LIN {X 0,Y 354.792,Z 356.911,A -85,B 0,C 180,E1 -13288.404,E2 -13288.404} C_VEL
LIN {X 0,Y 354.852,Z 356.899,A -85,B 0,C 180,E1 -13291.619,E2 -13291.619} C_VEL
LIN {X 0,Y 354.898,Z 356.892,A -85,B 0,C 180,E1 -13294.172,E2 -13294.172} C_VEL
LIN {X 0,Y 354.833,Z 356.903,A -85,B 0,C 180,E1 -13297.894,E2 -13297.894} C_VEL
LIN {X 0,Y 354.92,Z 356.896,A -85,B 0,C 180,E1 -13301.891,E2 -13301.891} C_VEL
LIN {X 0,Y 354.941,Z 356.88,A -85,B 0,C 180,E1 -13305.98,E2 -13305.98} C_VEL
LIN {X 0,Y 354.981,Z 356.892,A -85,B 0,C 180,E1 -13309.736,E2 -13309.736} C_VEL
LIN {X 0,Y 355.112,Z 356.874,A -85,B 0,C 180,E1 -13312.037,E2 -13312.037} C_VEL
LIN {X 0,Y 355.091,Z 356.88,A -85,B 0,C 180,E1 -13314.321,E2 -13314.321} C_VEL
LIN {X 0,Y 355.244,Z 356.86,A -85,B 0,C 180,E1 -13317.732,E2 -13317.732} C_VEL
LIN {X 0,Y 355.395,Z 356.843,A -85,B 0,C 180,E1 -13320,E2 -13320} C_VEL
LIN {X 0,Y 355.244,Z 356.859,A -85,B 0,C 180,E1 -13322.267,E2 -13322.267} C_VEL
LIN {X 0,Y 355.136,Z 356.874,A -85,B 0,C 180,E1 -13326.819,E2 -13326.819} C_VEL
LIN {X 0,Y 355.013,Z 356.89,A -85,B 0,C 180,E1 -13329.112,E2 -13329.112} C_VEL
LIN {X 0,Y 354.919,Z 356.896,A -85,B 0,C 180,E1 -13332.581,E2 -13332.581} C_VEL
LIN {X 0,Y 354.887,Z 356.902,A -85,B 0,C 180,E1 -13336.096,E2 -13336.096} C_VEL
LIN {X 0,Y 354.904,Z 356.9,A -85,B 0,C 180,E1 -13338.472,E2 -13338.472} C_VEL
LIN {X 0,Y 354.832,Z 356.911,A -85,B 0,C 180,E1 -13342.106,E2 -13342.106} C_VEL
LIN {X 0,Y 354.897,Z 356.906,A -85,B 0,C 180,E1 -13345.827,E2 -13345.827} C_VEL
LIN {X 0,Y 354.852,Z 356.911,A -85,B 0,C 180,E1 -13349.679,E2 -13349.679} C_VEL
LIN {X 0,Y 354.803,Z 356.914,A -85,B 0,C 180,E1 -13353.702,E2 -13353.702} C_VEL
LIN {X 0,Y 354.851,Z 357.111,A -85,B 0,C 180,E1 -13355.707,E2 -13355.707} C_VEL
LIN {X 0,Y 355.545,Z 361.082,A -85,B 0,C 180,E1 -13359.238,E2 -13359.238} C_VEL
LIN {X 0,Y 356.332,Z 365.897,A -85,B 0,C 180,E1 -13363.135,E2 -13363.135} C_VEL
LIN {X 0,Y 357.017,Z 370.347,A -85,B 0,C 180,E1 -13366.451,E2 -13366.451} C_VEL
LIN {X 0,Y 357.144,Z 373.14,A -85,B 0,C 180,E1 -13368.398,E2 -13368.398} C_VEL
LIN {X 0,Y 356.7,Z 376.988,A -85,B 0,C 180,E1 -13370.914,E2 -13370.914} C_VEL
LIN {X 0,Y 356.204,Z 381.837,A -85,B 0,C 180,E1 -13373.992,E2 -13373.992} C_VEL
LIN {X 0,Y 355.641,Z 386.853,A -85,B 0,C 180,E1 -13377.082,E2 -13377.082} C_VEL
LIN {X 0,Y 354.999,Z 392.89,A -85,B 0,C 180,E1 -13380.747,E2 -13380.747} C_VEL
LIN {X 0,Y 356.577,Z 398.562,A -85,B 0,C 180,E1 -13381.035,E2 -13381.035} C_VEL
LIN {X 0,Y 360.847,Z 413.008,A -85,B 0,C 180,E1 -13381.89,E2 -13381.89} C_VEL
LIN {X 0,Y 364.022,Z 427.002,A -85,B 0,C 180,E1 -13382.822,E2 -13382.822} C_VEL
LIN {X 0,Y 366.355,Z 441.422,A -85,B 0,C 180,E1 -13383.916,E2 -13383.916} C_VEL
LIN {X 0,Y 366.773,Z 446.491,A -85,B 0,C 180,E1 -13384.331,E2 -13384.331} C_VEL
LIN {X 0,Y 365.079,Z 460.119,A -85,B 0,C 180,E1 -13385.4,E2 -13385.4} C_VEL
LIN {X 0,Y 363.21,Z 472.884,A -85,B 0,C 180,E1 -13386.63,E2 -13386.63} C_VEL
LIN {X 0,Y 361.147,Z 485.804,A -85,B 0,C 180,E1 -13388.151,E2 -13388.151} C_VEL
LIN {X 0,Y 359.279,Z 497.794,A -85,B 0,C 180,E1 -13389.875,E2 -13389.875} C_VEL
LIN {X 0,Y 357.694,Z 508.176,A -85,B 0,C 180,E1 -13391.678,E2 -13391.678} C_VEL
LIN {X 0,Y 356.178,Z 517.746,A -85,B 0,C 180,E1 -13393.67,E2 -13393.67} C_VEL
LIN {X 0,Y 355.076,Z 525.736,A -85,B 0,C 180,E1 -13395.677,E2 -13395.677} C_VEL
LIN {X 0,Y 354.215,Z 533.203,A -85,B 0,C 180,E1 -13397.976,E2 -13397.976} C_VEL
LIN {X 0,Y 353.613,Z 539.134,A -85,B 0,C 180,E1 -13400.275,E2 -13400.275} C_VEL
LIN {X 0,Y 353.433,Z 542.669,A -85,B 0,C 180,E1 -13401.999,E2 -13401.999} C_VEL
LIN {X 0,Y 353.28,Z 546.243,A -85,B 0,C 180,E1 -13404.292,E2 -13404.292} C_VEL
LIN {X 0,Y 353.246,Z 548.596,A -85,B 0,C 180,E1 -13406.579,E2 -13406.579} C_VEL
LIN {X 0,Y 353.373,Z 549.786,A -85,B 0,C 180,E1 -13408.861,E2 -13408.861} C_VEL
LIN {X 0,Y 353.373,Z 549.784,A -85,B 0,C 180,E1 -13411.14,E2 -13411.14} C_VEL
LIN {X 0,Y 353.25,Z 548.585,A -85,B 0,C 180,E1 -13413.422,E2 -13413.422} C_VEL
LIN {X 0,Y 353.33,Z 546.227,A -85,B 0,C 180,E1 -13415.708,E2 -13415.708} C_VEL
LIN {X 0,Y 353.435,Z 542.651,A -85,B 0,C 180,E1 -13418.002,E2 -13418.002} C_VEL
LIN {X 0,Y 353.692,Z 537.771,A -85,B 0,C 180,E1 -13420.302,E2 -13420.302} C_VEL
LIN {X 0,Y 354.381,Z 531.47,A -85,B 0,C 180,E1 -13422.601,E2 -13422.601} C_VEL
LIN {X 0,Y 355.367,Z 523.568,A -85,B 0,C 180,E1 -13424.898,E2 -13424.898} C_VEL
LIN {X 0,Y 356.555,Z 515.174,A -85,B 0,C 180,E1 -13426.902,E2 -13426.902} C_VEL
LIN {X 0,Y 358.192,Z 505.081,A -85,B 0,C 180,E1 -13428.89,E2 -13428.89} C_VEL
LIN {X 0,Y 359.777,Z 494.765,A -85,B 0,C 180,E1 -13430.587,E2 -13430.587} C_VEL
LIN {X 0,Y 361.699,Z 482.486,A -85,B 0,C 180,E1 -13432.266,E2 -13432.266} C_VEL
LIN {X 0,Y 363.774,Z 468.83,A -85,B 0,C 180,E1 -13433.785,E2 -13433.785} C_VEL
LIN {X 0,Y 365.735,Z 455.151,A -85,B 0,C 180,E1 -13435.009,E2 -13435.009} C_VEL
LIN {X 0,Y 366.764,Z 445.121,A -85,B 0,C 180,E1 -13435.76,E2 -13435.76} C_VEL
LIN {X 0,Y 364.758,Z 431.05,A -85,B 0,C 180,E1 -13436.869,E2 -13436.869} C_VEL
LIN {X 0,Y 361.626,Z 416.135,A -85,B 0,C 180,E1 -13437.898,E2 -13437.898} C_VEL
LIN {X 0,Y 357.697,Z 401.937,A -85,B 0,C 180,E1 -13438.761,E2 -13438.761} C_VEL
LIN {X 0,Y 355.006,Z 392.859,A -85,B 0,C 180,E1 -13439.255,E2 -13439.255} C_VEL
LIN {X 0,Y 355.62,Z 386.82,A -85,B 0,C 180,E1 -13442.921,E2 -13442.921} C_VEL
LIN {X 0,Y 356.167,Z 381.789,A -85,B 0,C 180,E1 -13445.999,E2 -13445.999} C_VEL
LIN {X 0,Y 356.829,Z 375.826,A -85,B 0,C 180,E1 -13449.814,E2 -13449.814} C_VEL
LIN {X 0,Y 357.151,Z 372.485,A -85,B 0,C 180,E1 -13451.994,E2 -13451.994} C_VEL
LIN {X 0,Y 356.778,Z 368.497,A -85,B 0,C 180,E1 -13454.835,E2 -13454.835} C_VEL
LIN {X 0,Y 356.1,Z 364.541,A -85,B 0,C 180,E1 -13457.854,E2 -13457.854} C_VEL
LIN {X 0,Y 355.553,Z 361.02,A -85,B 0,C 180,E1 -13460.764,E2 -13460.764} C_VEL
LIN {X 0,Y 354.841,Z 356.914,A -85,B 0,C 180,E1 -13464.509,E2 -13464.509} C_VEL
LIN {X 0,Y 354.789,Z 356.916,A -85,B 0,C 180,E1 -13467.667,E2 -13467.667} C_VEL
LIN {X 0,Y 354.849,Z 356.91,A -85,B 0,C 180,E1 -13471.619,E2 -13471.619} C_VEL
LIN {X 0,Y 354.902,Z 356.905,A -85,B 0,C 180,E1 -13474.173,E2 -13474.173} C_VEL
LIN {X 0,Y 354.837,Z 356.911,A -85,B 0,C 180,E1 -13477.894,E2 -13477.894} C_VEL
LIN {X 0,Y 354.926,Z 356.901,A -85,B 0,C 180,E1 -13481.892,E2 -13481.892} C_VEL
LIN {X 0,Y 354.946,Z 356.901,A -85,B 0,C 180,E1 -13485.981,E2 -13485.981} C_VEL
LIN {X 0,Y 354.981,Z 356.895,A -85,B 0,C 180,E1 -13489.736,E2 -13489.736} C_VEL
LIN {X 0,Y 355.118,Z 356.879,A -85,B 0,C 180,E1 -13492.037,E2 -13492.037} C_VEL
LIN {X 0,Y 355.096,Z 356.878,A -85,B 0,C 180,E1 -13494.321,E2 -13494.321} C_VEL
LIN {X 0,Y 355.249,Z 356.858,A -85,B 0,C 180,E1 -13497.733,E2 -13497.733} C_VEL
LIN {X 0,Y 355.399,Z 356.838,A -85,B 0,C 180,E1 -13500,E2 -13500} C_VEL
LIN {X 0,Y 355.249,Z 356.858,A -85,B 0,C 180,E1 -13502.268,E2 -13502.268} C_VEL
LIN {X 0,Y 355.142,Z 356.868,A -85,B 0,C 180,E1 -13506.819,E2 -13506.819} C_VEL
LIN {X 0,Y 355.019,Z 356.888,A -85,B 0,C 180,E1 -13509.112,E2 -13509.112} C_VEL
LIN {X 0,Y 354.924,Z 356.873,A -85,B 0,C 180,E1 -13512.581,E2 -13512.581} C_VEL
LIN {X 0,Y 354.893,Z 356.901,A -85,B 0,C 180,E1 -13516.096,E2 -13516.096} C_VEL
LIN {X 0,Y 354.905,Z 356.894,A -85,B 0,C 180,E1 -13518.472,E2 -13518.472} C_VEL
LIN {X 0,Y 354.83,Z 356.902,A -85,B 0,C 180,E1 -13522.106,E2 -13522.106} C_VEL
LIN {X 0,Y 354.902,Z 356.893,A -85,B 0,C 180,E1 -13525.827,E2 -13525.827} C_VEL
LIN {X 0,Y 354.821,Z 356.91,A -85,B 0,C 180,E1 -13529.682,E2 -13529.682} C_VEL
LIN {X 0,Y 354.809,Z 356.9,A -85,B 0,C 180,E1 -13533.702,E2 -13533.702} C_VEL
LIN {X 0,Y 354.802,Z 356.917,A -85,B 0,C 180,E1 -13536.459,E2 -13536.459} C_VEL
LIN {X 0,Y 354.827,Z 356.912,A -85,B 0,C 180,E1 -13539.423,E2 -13539.423} C_VEL
LIN {X 0,Y 354.791,Z 356.918,A -85,B 0,C 180,E1 -13542.867,E2 -13542.867} C_VEL
LIN {X 0,Y 354.759,Z 356.925,A -85,B 0,C 180,E1 -13546.102,E2 -13546.102} C_VEL
LIN {X 0,Y 354.646,Z 356.938,A -85,B 0,C 180,E1 -13549.159,E2 -13549.159} C_VEL
LIN {X 0,Y 354.551,Z 356.949,A -85,B 0,C 180,E1 -13550.63,E2 -13550.63} C_VEL
LIN {X 0,Y 354.388,Z 358.655,A -85,B 0,C 180,E1 -13553.491,E2 -13553.491} C_VEL
LIN {X 0,Y 354.329,Z 360.804,A -85,B 0,C 180,E1 -13556.414,E2 -13556.414} C_VEL
LIN {X 0,Y 354.246,Z 362.804,A -85,B 0,C 180,E1 -13558.947,E2 -13558.947} C_VEL
LIN {X 0,Y 354.18,Z 364.301,A -85,B 0,C 180,E1 -13560.767,E2 -13560.767} C_VEL
LIN {X 0,Y 355.13,Z 367.269,A -85,B 0,C 180,E1 -13560.946,E2 -13560.946} C_VEL
LIN {X 0,Y 360.606,Z 380.429,A -85,B 0,C 180,E1 -13561.869,E2 -13561.869} C_VEL
LIN {X 0,Y 365.001,Z 393.413,A -85,B 0,C 180,E1 -13562.86,E2 -13562.86} C_VEL
LIN {X 0,Y 368.598,Z 406.777,A -85,B 0,C 180,E1 -13563.989,E2 -13563.989} C_VEL
LIN {X 0,Y 367.247,Z 420.846,A -85,B 0,C 180,E1 -13564.996,E2 -13564.996} C_VEL
LIN {X 0,Y 365.75,Z 432.854,A -85,B 0,C 180,E1 -13566.051,E2 -13566.051} C_VEL
LIN {X 0,Y 363.869,Z 445.767,A -85,B 0,C 180,E1 -13567.425,E2 -13567.425} C_VEL
LIN {X 0,Y 362.072,Z 457.604,A -85,B 0,C 180,E1 -13568.965,E2 -13568.965} C_VEL
LIN {X 0,Y 360.34,Z 468.309,A -85,B 0,C 180,E1 -13570.636,E2 -13570.636} C_VEL
LIN {X 0,Y 358.782,Z 477.435,A -85,B 0,C 180,E1 -13572.324,E2 -13572.324} C_VEL
LIN {X 0,Y 357.29,Z 486.251,A -85,B 0,C 180,E1 -13574.283,E2 -13574.283} C_VEL
LIN {X 0,Y 356.202,Z 493.723,A -85,B 0,C 180,E1 -13576.304,E2 -13576.304} C_VEL
LIN {X 0,Y 355.03,Z 500.622,A -85,B 0,C 180,E1 -13578.582,E2 -13578.582} C_VEL
LIN {X 0,Y 354.333,Z 506.03,A -85,B 0,C 180,E1 -13580.869,E2 -13580.869} C_VEL
LIN {X 0,Y 353.792,Z 510.388,A -85,B 0,C 180,E1 -13583.335,E2 -13583.335} C_VEL
LIN {X 0,Y 353.521,Z 512.977,A -85,B 0,C 180,E1 -13585.439,E2 -13585.439} C_VEL
LIN {X 0,Y 353.488,Z 514.694,A -85,B 0,C 180,E1 -13587.721,E2 -13587.721} C_VEL
LIN {X 0,Y 353.421,Z 515.297,A -85,B 0,C 180,E1 -13590,E2 -13590} C_VEL
LIN {X 0,Y 353.488,Z 514.739,A -85,B 0,C 180,E1 -13592.278,E2 -13592.278} C_VEL
LIN {X 0,Y 353.52,Z 513.08,A -85,B 0,C 180,E1 -13594.561,E2 -13594.561} C_VEL
LIN {X 0,Y 353.803,Z 510.271,A -85,B 0,C 180,E1 -13596.845,E2 -13596.845} C_VEL
LIN {X 0,Y 354.289,Z 506.244,A -85,B 0,C 180,E1 -13599.131,E2 -13599.131} C_VEL
LIN {X 0,Y 354.996,Z 500.903,A -85,B 0,C 180,E1 -13601.418,E2 -13601.418} C_VEL
LIN {X 0,Y 356.098,Z 494.084,A -85,B 0,C 180,E1 -13603.699,E2 -13603.699} C_VEL
LIN {X 0,Y 357.197,Z 486.711,A -85,B 0,C 180,E1 -13605.707,E2 -13605.707} C_VEL
LIN {X 0,Y 358.711,Z 477.904,A -85,B 0,C 180,E1 -13607.678,E2 -13607.678} C_VEL
LIN {X 0,Y 360.259,Z 468.873,A -85,B 0,C 180,E1 -13609.368,E2 -13609.368} C_VEL
LIN {X 0,Y 362.038,Z 457.697,A -85,B 0,C 180,E1 -13611.126,E2 -13611.126} C_VEL
LIN {X 0,Y 363.94,Z 445.402,A -85,B 0,C 180,E1 -13612.719,E2 -13612.719} C_VEL
LIN {X 0,Y 365.804,Z 432.419,A -85,B 0,C 180,E1 -13614.095,E2 -13614.095} C_VEL
LIN {X 0,Y 367.449,Z 419.304,A -85,B 0,C 180,E1 -13615.226,E2 -13615.226} C_VEL
LIN {X 0,Y 368.586,Z 406.514,A -85,B 0,C 180,E1 -13616.133,E2 -13616.133} C_VEL
LIN {X 0,Y 364.62,Z 392.07,A -85,B 0,C 180,E1 -13617.345,E2 -13617.345} C_VEL
LIN {X 0,Y 359.758,Z 378.332,A -85,B 0,C 180,E1 -13618.393,E2 -13618.393} C_VEL
LIN {X 0,Y 354.941,Z 366.959,A -85,B 0,C 180,E1 -13619.187,E2 -13619.187} C_VEL
LIN {X 0,Y 354.127,Z 364.27,A -85,B 0,C 180,E1 -13619.354,E2 -13619.354} C_VEL
LIN {X 0,Y 354.277,Z 361.813,A -85,B 0,C 180,E1 -13622.385,E2 -13622.385} C_VEL
LIN {X 0,Y 354.282,Z 361.372,A -85,B 0,C 180,E1 -13622.97,E2 -13622.97} C_VEL
LIN {X 0,Y 353.664,Z 360.751,A -85,B 0,C 180,E1 -13623.914,E2 -13623.914} C_VEL
LIN {X 0,Y 350.891,Z 359.984,A -85,B 0,C 180,E1 -13625.456,E2 -13625.456} C_VEL
LIN {X 0,Y 348.521,Z 359.395,A -85,B 0,C 180,E1 -13626.703,E2 -13626.703} C_VEL
LIN {X 0,Y 347.502,Z 358.841,A -85,B 0,C 180,E1 -13627.666,E2 -13627.666} C_VEL
LIN {X 0,Y 347.418,Z 358.622,A -85,B 0,C 180,E1 -13627.991,E2 -13627.991} C_VEL
LIN {X 0,Y 347.444,Z 358.029,A -85,B 0,C 180,E1 -13628.833,E2 -13628.833} C_VEL
LIN {X 0,Y 347.67,Z 357.799,A -85,B 0,C 180,E1 -13631.841,E2 -13631.841} C_VEL
LIN {X 0,Y 347.702,Z 357.799,A -85,B 0,C 180,E1 -13635.027,E2 -13635.027} C_VEL
LIN {X 0,Y 347.749,Z 357.793,A -85,B 0,C 180,E1 -13638.397,E2 -13638.397} C_VEL
LIN {X 0,Y 347.773,Z 357.791,A -85,B 0,C 180,E1 -13642.011,E2 -13642.011} C_VEL
LIN {X 0,Y 347.743,Z 357.789,A -85,B 0,C 180,E1 -13645.536,E2 -13645.536} C_VEL
LIN {X 0,Y 347.762,Z 357.793,A -85,B 0,C 180,E1 -13649.653,E2 -13649.653} C_VEL
LIN {X 0,Y 347.851,Z 357.763,A -85,B 0,C 180,E1 -13652.744,E2 -13652.744} C_VEL
LIN {X 0,Y 347.787,Z 357.788,A -85,B 0,C 180,E1 -13656.162,E2 -13656.162} C_VEL
LIN {X 0,Y 347.81,Z 357.764,A -85,B 0,C 180,E1 -13659.909,E2 -13659.909} C_VEL
LIN {X 0,Y 347.864,Z 357.778,A -85,B 0,C 180,E1 -13662.359,E2 -13662.359} C_VEL
LIN {X 0,Y 347.895,Z 357.757,A -85,B 0,C 180,E1 -13665.971,E2 -13665.971} C_VEL
LIN {X 0,Y 347.931,Z 357.767,A -85,B 0,C 180,E1 -13669.526,E2 -13669.526} C_VEL
LIN {X 0,Y 348.072,Z 357.751,A -85,B 0,C 180,E1 -13671.875,E2 -13671.875} C_VEL
LIN {X 0,Y 348.066,Z 357.755,A -85,B 0,C 180,E1 -13674.206,E2 -13674.206} C_VEL
LIN {X 0,Y 348.206,Z 357.737,A -85,B 0,C 180,E1 -13677.686,E2 -13677.686} C_VEL
LIN {X 0,Y 348.365,Z 357.719,A -85,B 0,C 180,E1 -13680,E2 -13680} C_VEL
LIN {X 0,Y 348.207,Z 357.736,A -85,B 0,C 180,E1 -13682.313,E2 -13682.313} C_VEL
LIN {X 0,Y 348.104,Z 357.749,A -85,B 0,C 180,E1 -13686.958,E2 -13686.958} C_VEL
LIN {X 0,Y 347.965,Z 357.769,A -85,B 0,C 180,E1 -13689.298,E2 -13689.298} C_VEL
LIN {X 0,Y 347.888,Z 357.772,A -85,B 0,C 180,E1 -13692.839,E2 -13692.839} C_VEL
LIN {X 0,Y 347.837,Z 357.78,A -85,B 0,C 180,E1 -13696.431,E2 -13696.431} C_VEL
LIN {X 0,Y 347.853,Z 357.78,A -85,B 0,C 180,E1 -13698.86,E2 -13698.86} C_VEL
LIN {X 0,Y 347.772,Z 357.791,A -85,B 0,C 180,E1 -13702.579,E2 -13702.579} C_VEL
LIN {X 0,Y 347.81,Z 357.788,A -85,B 0,C 180,E1 -13705.108,E2 -13705.108} C_VEL
LIN {X 0,Y 347.81,Z 357.79,A -85,B 0,C 180,E1 -13707.694,E2 -13707.694} C_VEL
LIN {X 0,Y 347.762,Z 357.794,A -85,B 0,C 180,E1 -13710.347,E2 -13710.347} C_VEL
LIN {X 0,Y 347.742,Z 357.797,A -85,B 0,C 180,E1 -13714.464,E2 -13714.464} C_VEL
LIN {X 0,Y 347.821,Z 357.98,A -85,B 0,C 180,E1 -13715.16,E2 -13715.16} C_VEL
LIN {X 0,Y 348.464,Z 361.88,A -85,B 0,C 180,E1 -13718.698,E2 -13718.698} C_VEL
LIN {X 0,Y 349.074,Z 365.588,A -85,B 0,C 180,E1 -13721.848,E2 -13721.848} C_VEL
LIN {X 0,Y 349.84,Z 370.026,A -85,B 0,C 180,E1 -13725.323,E2 -13725.323} C_VEL
LIN {X 0,Y 350.146,Z 373.663,A -85,B 0,C 180,E1 -13727.958,E2 -13727.958} C_VEL
LIN {X 0,Y 349.709,Z 377.764,A -85,B 0,C 180,E1 -13730.726,E2 -13730.726} C_VEL
LIN {X 0,Y 349.092,Z 383.238,A -85,B 0,C 180,E1 -13734.28,E2 -13734.28} C_VEL
LIN {X 0,Y 348.473,Z 388.953,A -85,B 0,C 180,E1 -13737.893,E2 -13737.893} C_VEL
LIN {X 0,Y 348.058,Z 392.505,A -85,B 0,C 180,E1 -13740.097,E2 -13740.097} C_VEL
LIN {X 0,Y 348.978,Z 395.921,A -85,B 0,C 180,E1 -13740.281,E2 -13740.281} C_VEL
LIN {X 0,Y 353.632,Z 411.282,A -85,B 0,C 180,E1 -13741.205,E2 -13741.205} C_VEL
LIN {X 0,Y 357.038,Z 425.815,A -85,B 0,C 180,E1 -13742.197,E2 -13742.197} C_VEL
LIN {X 0,Y 359.373,Z 439.628,A -85,B 0,C 180,E1 -13743.27,E2 -13743.27} C_VEL
LIN {X 0,Y 360.234,Z 446.964,A -85,B 0,C 180,E1 -13743.894,E2 -13743.894} C_VEL
LIN {X 0,Y 358.379,Z 461.362,A -85,B 0,C 180,E1 -13745.063,E2 -13745.063} C_VEL
LIN {X 0,Y 356.448,Z 473.835,A -85,B 0,C 180,E1 -13746.314,E2 -13746.314} C_VEL
LIN {X 0,Y 354.316,Z 486.533,A -85,B 0,C 180,E1 -13747.86,E2 -13747.86} C_VEL
LIN {X 0,Y 352.389,Z 498.32,A -85,B 0,C 180,E1 -13749.613,E2 -13749.613} C_VEL
LIN {X 0,Y 350.889,Z 507.826,A -85,B 0,C 180,E1 -13751.309,E2 -13751.309} C_VEL
LIN {X 0,Y 349.288,Z 517.396,A -85,B 0,C 180,E1 -13753.339,E2 -13753.339} C_VEL
LIN {X 0,Y 348.092,Z 525.588,A -85,B 0,C 180,E1 -13755.442,E2 -13755.442} C_VEL
LIN {X 0,Y 347.202,Z 532.853,A -85,B 0,C 180,E1 -13757.729,E2 -13757.729} C_VEL
LIN {X 0,Y 346.555,Z 538.784,A -85,B 0,C 180,E1 -13760.074,E2 -13760.074} C_VEL
LIN {X 0,Y 346.358,Z 542.32,A -85,B 0,C 180,E1 -13761.835,E2 -13761.835} C_VEL
LIN {X 0,Y 346.199,Z 545.895,A -85,B 0,C 180,E1 -13764.175,E2 -13764.175} C_VEL
LIN {X 0,Y 346.168,Z 548.249,A -85,B 0,C 180,E1 -13766.509,E2 -13766.509} C_VEL
LIN {X 0,Y 346.276,Z 549.438,A -85,B 0,C 180,E1 -13768.838,E2 -13768.838} C_VEL
LIN {X 0,Y 346.276,Z 549.436,A -85,B 0,C 180,E1 -13771.163,E2 -13771.163} C_VEL
LIN {X 0,Y 346.172,Z 548.237,A -85,B 0,C 180,E1 -13773.492,E2 -13773.492} C_VEL
LIN {X 0,Y 346.286,Z 545.621,A -85,B 0,C 180,E1 -13776.028,E2 -13776.028} C_VEL
LIN {X 0,Y 346.418,Z 541.213,A -85,B 0,C 180,E1 -13778.752,E2 -13778.752} C_VEL
LIN {X 0,Y 346.835,Z 535.971,A -85,B 0,C 180,E1 -13781.099,E2 -13781.099} C_VEL
LIN {X 0,Y 347.596,Z 529.278,A -85,B 0,C 180,E1 -13783.446,E2 -13783.446} C_VEL
LIN {X 0,Y 348.579,Z 522.082,A -85,B 0,C 180,E1 -13785.495,E2 -13785.495} C_VEL
LIN {X 0,Y 349.86,Z 513.45,A -85,B 0,C 180,E1 -13787.537,E2 -13787.537} C_VEL
LIN {X 0,Y 351.651,Z 503.082,A -85,B 0,C 180,E1 -13789.558,E2 -13789.558} C_VEL
LIN {X 0,Y 353.364,Z 492.483,A -85,B 0,C 180,E1 -13791.283,E2 -13791.283} C_VEL
LIN {X 0,Y 355.241,Z 480.973,A -85,B 0,C 180,E1 -13792.846,E2 -13792.846} C_VEL
LIN {X 0,Y 357.257,Z 468.476,A -85,B 0,C 180,E1 -13794.246,E2 -13794.246} C_VEL
LIN {X 0,Y 359.281,Z 454.797,A -85,B 0,C 180,E1 -13795.49,E2 -13795.49} C_VEL
LIN {X 0,Y 360.162,Z 446.23,A -85,B 0,C 180,E1 -13796.153,E2 -13796.153} C_VEL
LIN {X 0,Y 358.311,Z 432.718,A -85,B 0,C 180,E1 -13797.27,E2 -13797.27} C_VEL
LIN {X 0,Y 355.067,Z 416.892,A -85,B 0,C 180,E1 -13798.41,E2 -13798.41} C_VEL
LIN {X 0,Y 350.843,Z 401.801,A -85,B 0,C 180,E1 -13799.37,E2 -13799.37} C_VEL
LIN {X 0,Y 348.151,Z 393.412,A -85,B 0,C 180,E1 -13799.842,E2 -13799.842} C_VEL
LIN {X 0,Y 348.047,Z 392.512,A -85,B 0,C 180,E1 -13799.884,E2 -13799.884} C_VEL
LIN {X 0,Y 348.861,Z 385.406,A -85,B 0,C 180,E1 -13804.314,E2 -13804.314} C_VEL
LIN {X 0,Y 349.519,Z 379.113,A -85,B 0,C 180,E1 -13808.354,E2 -13808.354} C_VEL
LIN {X 0,Y 350.121,Z 374.414,A -85,B 0,C 180,E1 -13811.485,E2 -13811.485} C_VEL
LIN {X 0,Y 350,Z 371.261,A -85,B 0,C 180,E1 -13813.707,E2 -13813.707} C_VEL
LIN {X 0,Y 349.36,Z 367.126,A -85,B 0,C 180,E1 -13816.845,E2 -13816.845} C_VEL
LIN {X 0,Y 348.741,Z 363.333,A -85,B 0,C 180,E1 -13819.978,E2 -13819.978} C_VEL
LIN {X 0,Y 347.99,Z 358.928,A -85,B 0,C 180,E1 -13823.886,E2 -13823.886} C_VEL
LIN {X 0,Y 347.78,Z 357.796,A -85,B 0,C 180,E1 -13825.189,E2 -13825.189} C_VEL
LIN {X 0,Y 347.747,Z 357.796,A -85,B 0,C 180,E1 -13828.301,E2 -13828.301} C_VEL
LIN {X 0,Y 347.781,Z 357.791,A -85,B 0,C 180,E1 -13830.988,E2 -13830.988} C_VEL
LIN {X 0,Y 347.834,Z 357.785,A -85,B 0,C 180,E1 -13833.608,E2 -13833.608} C_VEL
LIN {X 0,Y 347.791,Z 357.788,A -85,B 0,C 180,E1 -13836.162,E2 -13836.162} C_VEL
LIN {X 0,Y 347.82,Z 357.786,A -85,B 0,C 180,E1 -13839.91,E2 -13839.91} C_VEL
LIN {X 0,Y 347.869,Z 357.779,A -85,B 0,C 180,E1 -13842.36,E2 -13842.36} C_VEL
LIN {X 0,Y 347.9,Z 357.779,A -85,B 0,C 180,E1 -13845.971,E2 -13845.971} C_VEL
LIN {X 0,Y 347.932,Z 357.774,A -85,B 0,C 180,E1 -13849.526,E2 -13849.526} C_VEL
LIN {X 0,Y 348.078,Z 357.755,A -85,B 0,C 180,E1 -13851.875,E2 -13851.875} C_VEL
LIN {X 0,Y 348.071,Z 357.754,A -85,B 0,C 180,E1 -13854.206,E2 -13854.206} C_VEL
LIN {X 0,Y 348.211,Z 357.735,A -85,B 0,C 180,E1 -13857.687,E2 -13857.687} C_VEL
LIN {X 0,Y 348.348,Z 357.716,A -85,B 0,C 180,E1 -13860,E2 -13860} C_VEL
LIN {X 0,Y 348.211,Z 357.735,A -85,B 0,C 180,E1 -13862.314,E2 -13862.314} C_VEL
LIN {X 0,Y 348.11,Z 357.744,A -85,B 0,C 180,E1 -13866.958,E2 -13866.958} C_VEL
LIN {X 0,Y 347.971,Z 357.765,A -85,B 0,C 180,E1 -13869.299,E2 -13869.299} C_VEL
LIN {X 0,Y 347.893,Z 357.747,A -85,B 0,C 180,E1 -13872.839,E2 -13872.839} C_VEL
LIN {X 0,Y 347.843,Z 357.781,A -85,B 0,C 180,E1 -13876.431,E2 -13876.431} C_VEL
LIN {X 0,Y 347.854,Z 357.771,A -85,B 0,C 180,E1 -13878.86,E2 -13878.86} C_VEL
LIN {X 0,Y 347.771,Z 357.784,A -85,B 0,C 180,E1 -13882.58,E2 -13882.58} C_VEL
LIN {X 0,Y 347.815,Z 357.782,A -85,B 0,C 180,E1 -13885.108,E2 -13885.108} C_VEL
LIN {X 0,Y 347.811,Z 357.768,A -85,B 0,C 180,E1 -13887.694,E2 -13887.694} C_VEL
LIN {X 0,Y 347.752,Z 357.795,A -85,B 0,C 180,E1 -13890.348,E2 -13890.348} C_VEL
LIN {X 0,Y 347.751,Z 357.781,A -85,B 0,C 180,E1 -13894.044,E2 -13894.044} C_VEL
LIN {X 0,Y 347.766,Z 357.791,A -85,B 0,C 180,E1 -13897.32,E2 -13897.32} C_VEL
LIN {X 0,Y 347.736,Z 357.796,A -85,B 0,C 180,E1 -13900.297,E2 -13900.297} C_VEL
LIN {X 0,Y 347.726,Z 357.798,A -85,B 0,C 180,E1 -13903.408,E2 -13903.408} C_VEL
LIN {X 0,Y 347.718,Z 357.803,A -85,B 0,C 180,E1 -13906.688,E2 -13906.688} C_VEL
LIN {X 0,Y 347.551,Z 357.821,A -85,B 0,C 180,E1 -13909.677,E2 -13909.677} C_VEL
LIN {X 0,Y 347.443,Z 357.947,A -85,B 0,C 180,E1 -13911.166,E2 -13911.166} C_VEL
LIN {X 0,Y 347.335,Z 360.038,A -85,B 0,C 180,E1 -13914.07,E2 -13914.07} C_VEL
LIN {X 0,Y 347.266,Z 362.085,A -85,B 0,C 180,E1 -13916.877,E2 -13916.877} C_VEL
LIN {X 0,Y 347.132,Z 364.664,A -85,B 0,C 180,E1 -13920.105,E2 -13920.105} C_VEL
LIN {X 0,Y 348.332,Z 368.023,A -85,B 0,C 180,E1 -13920.333,E2 -13920.333} C_VEL
LIN {X 0,Y 353.964,Z 381.605,A -85,B 0,C 180,E1 -13921.328,E2 -13921.328} C_VEL
LIN {X 0,Y 358.362,Z 394.279,A -85,B 0,C 180,E1 -13922.34,E2 -13922.34} C_VEL
LIN {X 0,Y 361.801,Z 407.157,A -85,B 0,C 180,E1 -13923.463,E2 -13923.463} C_VEL
LIN {X 0,Y 362.156,Z 409.029,A -85,B 0,C 180,E1 -13923.623,E2 -13923.623} C_VEL
LIN {X 0,Y 360.697,Z 422.417,A -85,B 0,C 180,E1 -13924.617,E2 -13924.617} C_VEL
LIN {X 0,Y 359.104,Z 434.623,A -85,B 0,C 180,E1 -13925.733,E2 -13925.733} C_VEL
LIN {X 0,Y 357.148,Z 447.283,A -85,B 0,C 180,E1 -13927.129,E2 -13927.129} C_VEL
LIN {X 0,Y 355.539,Z 457.305,A -85,B 0,C 180,E1 -13928.456,E2 -13928.456} C_VEL
LIN {X 0,Y 353.901,Z 467.036,A -85,B 0,C 180,E1 -13929.966,E2 -13929.966} C_VEL
LIN {X 0,Y 351.994,Z 477.787,A -85,B 0,C 180,E1 -13931.972,E2 -13931.972} C_VEL
LIN {X 0,Y 350.429,Z 486.674,A -85,B 0,C 180,E1 -13933.985,E2 -13933.985} C_VEL
LIN {X 0,Y 349.268,Z 494.075,A -85,B 0,C 180,E1 -13936.026,E2 -13936.026} C_VEL
LIN {X 0,Y 348.053,Z 500.972,A -85,B 0,C 180,E1 -13938.35,E2 -13938.35} C_VEL
LIN {X 0,Y 347.309,Z 506.38,A -85,B 0,C 180,E1 -13940.683,E2 -13940.683} C_VEL
LIN {X 0,Y 346.717,Z 510.939,A -85,B 0,C 180,E1 -13943.333,E2 -13943.333} C_VEL
LIN {X 0,Y 346.46,Z 513.325,A -85,B 0,C 180,E1 -13945.345,E2 -13945.345} C_VEL
LIN {X 0,Y 346.395,Z 515.042,A -85,B 0,C 180,E1 -13947.674,E2 -13947.674} C_VEL
LIN {X 0,Y 346.341,Z 515.644,A -85,B 0,C 180,E1 -13950,E2 -13950} C_VEL
LIN {X 0,Y 346.395,Z 515.086,A -85,B 0,C 180,E1 -13952.325,E2 -13952.325} C_VEL
LIN {X 0,Y 346.459,Z 513.427,A -85,B 0,C 180,E1 -13954.654,E2 -13954.654} C_VEL
LIN {X 0,Y 346.746,Z 510.618,A -85,B 0,C 180,E1 -13956.985,E2 -13956.985} C_VEL
LIN {X 0,Y 347.276,Z 506.591,A -85,B 0,C 180,E1 -13959.317,E2 -13959.317} C_VEL
LIN {X 0,Y 348.021,Z 501.25,A -85,B 0,C 180,E1 -13961.65,E2 -13961.65} C_VEL
LIN {X 0,Y 349.174,Z 494.431,A -85,B 0,C 180,E1 -13963.976,E2 -13963.976} C_VEL
LIN {X 0,Y 350.336,Z 487.102,A -85,B 0,C 180,E1 -13966.011,E2 -13966.011} C_VEL
LIN {X 0,Y 351.939,Z 478.25,A -85,B 0,C 180,E1 -13968.03,E2 -13968.03} C_VEL
LIN {X 0,Y 353.528,Z 469.22,A -85,B 0,C 180,E1 -13969.752,E2 -13969.752} C_VEL
LIN {X 0,Y 355.345,Z 458.483,A -85,B 0,C 180,E1 -13971.474,E2 -13971.474} C_VEL
LIN {X 0,Y 357.213,Z 446.911,A -85,B 0,C 180,E1 -13973.018,E2 -13973.018} C_VEL
LIN {X 0,Y 359.179,Z 434.176,A -85,B 0,C 180,E1 -13974.415,E2 -13974.415} C_VEL
LIN {X 0,Y 360.738,Z 422.41,A -85,B 0,C 180,E1 -13975.486,E2 -13975.486} C_VEL
LIN {X 0,Y 362.161,Z 408.662,A -85,B 0,C 180,E1 -13976.508,E2 -13976.508} C_VEL
LIN {X 0,Y 358.206,Z 393.724,A -85,B 0,C 180,E1 -13977.808,E2 -13977.808} C_VEL
LIN {X 0,Y 352.975,Z 379.129,A -85,B 0,C 180,E1 -13978.974,E2 -13978.974} C_VEL
LIN {X 0,Y 348.071,Z 367.614,A -85,B 0,C 180,E1 -13979.812,E2 -13979.812} C_VEL
LIN {X 0,Y 347.116,Z 364.65,A -85,B 0,C 180,E1 -13979.995,E2 -13979.995} C_VEL
LIN {X 0,Y 347.26,Z 362.175,A -85,B 0,C 180,E1 -13983.122,E2 -13983.122} C_VEL
LIN {X 0,Y 347.339,Z 360.094,A -85,B 0,C 180,E1 -13985.967,E2 -13985.967} C_VEL
LIN {X 0,Y 347.418,Z 358.622,A -85,B 0,C 180,E1 -13987.991,E2 -13987.991} C_VEL
LIN {X 0,Y 346.776,Z 358.196,A -85,B 0,C 180,E1 -13988.956,E2 -13988.956} C_VEL
LIN {X 0,Y 344.046,Z 358.252,A -85,B 0,C 180,E1 -13990.537,E2 -13990.537} C_VEL
LIN {X 0,Y 341.728,Z 358.539,A -85,B 0,C 180,E1 -13991.819,E2 -13991.819} C_VEL
LIN {X 0,Y 340.727,Z 358.665,A -85,B 0,C 180,E1 -13992.808,E2 -13992.808} C_VEL
LIN {X 0,Y 340.641,Z 358.675,A -85,B 0,C 180,E1 -13993.143,E2 -13993.143} C_VEL
LIN {X 0,Y 340.674,Z 358.675,A -85,B 0,C 180,E1 -13997.095,E2 -13997.095} C_VEL
LIN {X 0,Y 340.697,Z 358.672,A -85,B 0,C 180,E1 -14000.247,E2 -14000.247} C_VEL
LIN {X 0,Y 340.709,Z 358.67,A -85,B 0,C 180,E1 -14003.559,E2 -14003.559} C_VEL
LIN {X 0,Y 340.692,Z 358.662,A -85,B 0,C 180,E1 -14006.153,E2 -14006.153} C_VEL
LIN {X 0,Y 340.773,Z 358.661,A -85,B 0,C 180,E1 -14010.332,E2 -14010.332} C_VEL
LIN {X 0,Y 340.803,Z 358.641,A -85,B 0,C 180,E1 -14013.02,E2 -14013.02} C_VEL
LIN {X 0,Y 340.727,Z 358.667,A -85,B 0,C 180,E1 -14016.927,E2 -14016.927} C_VEL
LIN {X 0,Y 340.788,Z 358.645,A -85,B 0,C 180,E1 -14020.733,E2 -14020.733} C_VEL
LIN {X 0,Y 340.785,Z 358.661,A -85,B 0,C 180,E1 -14023.218,E2 -14023.218} C_VEL
LIN {X 0,Y 340.845,Z 358.629,A -85,B 0,C 180,E1 -14026.89,E2 -14026.89} C_VEL
LIN {X 0,Y 340.928,Z 358.643,A -85,B 0,C 180,E1 -14030.508,E2 -14030.508} C_VEL
LIN {X 0,Y 341.074,Z 358.626,A -85,B 0,C 180,E1 -14032.898,E2 -14032.898} C_VEL
LIN {X 0,Y 341.168,Z 358.614,A -85,B 0,C 180,E1 -14037.639,E2 -14037.639} C_VEL
LIN {X 0,Y 341.314,Z 358.597,A -85,B 0,C 180,E1 -14040,E2 -14040} C_VEL
LIN {X 0,Y 341.168,Z 358.612,A -85,B 0,C 180,E1 -14042.361,E2 -14042.361} C_VEL
LIN {X 0,Y 341.074,Z 358.625,A -85,B 0,C 180,E1 -14047.102,E2 -14047.102} C_VEL
LIN {X 0,Y 340.869,Z 358.651,A -85,B 0,C 180,E1 -14050.694,E2 -14050.694} C_VEL
LIN {X 0,Y 340.86,Z 358.65,A -85,B 0,C 180,E1 -14054.325,E2 -14054.325} C_VEL
LIN {X 0,Y 340.835,Z 358.652,A -85,B 0,C 180,E1 -14058.467,E2 -14058.467} C_VEL
LIN {X 0,Y 340.751,Z 358.666,A -85,B 0,C 180,E1 -14061.857,E2 -14061.857} C_VEL
LIN {X 0,Y 340.77,Z 358.665,A -85,B 0,C 180,E1 -14065.664,E2 -14065.664} C_VEL
LIN {X 0,Y 340.74,Z 358.669,A -85,B 0,C 180,E1 -14068.32,E2 -14068.32} C_VEL
LIN {X 0,Y 340.702,Z 358.673,A -85,B 0,C 180,E1 -14071.044,E2 -14071.044} C_VEL
LIN {X 0,Y 340.72,Z 358.687,A -85,B 0,C 180,E1 -14074.405,E2 -14074.405} C_VEL
LIN {X 0,Y 341.413,Z 362.616,A -85,B 0,C 180,E1 -14078.137,E2 -14078.137} C_VEL
LIN {X 0,Y 341.963,Z 366.035,A -85,B 0,C 180,E1 -14081.122,E2 -14081.122} C_VEL
LIN {X 0,Y 342.79,Z 370.851,A -85,B 0,C 180,E1 -14085.018,E2 -14085.018} C_VEL
LIN {X 0,Y 343.109,Z 374.179,A -85,B 0,C 180,E1 -14087.51,E2 -14087.51} C_VEL
LIN {X 0,Y 342.959,Z 376.74,A -85,B 0,C 180,E1 -14089.307,E2 -14089.307} C_VEL
LIN {X 0,Y 342.213,Z 382.892,A -85,B 0,C 180,E1 -14093.447,E2 -14093.447} C_VEL
LIN {X 0,Y 341.725,Z 387.227,A -85,B 0,C 180,E1 -14096.27,E2 -14096.27} C_VEL
LIN {X 0,Y 341.12,Z 392.118,A -85,B 0,C 180,E1 -14099.421,E2 -14099.421} C_VEL
LIN {X 0,Y 342.974,Z 398.458,A -85,B 0,C 180,E1 -14099.787,E2 -14099.787} C_VEL
LIN {X 0,Y 347.532,Z 413.764,A -85,B 0,C 180,E1 -14100.777,E2 -14100.777} C_VEL
LIN {X 0,Y 350.783,Z 428.267,A -85,B 0,C 180,E1 -14101.829,E2 -14101.829} C_VEL
LIN {X 0,Y 353.076,Z 442.702,A -85,B 0,C 180,E1 -14103.015,E2 -14103.015} C_VEL
LIN {X 0,Y 353.623,Z 447.31,A -85,B 0,C 180,E1 -14103.424,E2 -14103.424} C_VEL
LIN {X 0,Y 351.933,Z 461.018,A -85,B 0,C 180,E1 -14104.574,E2 -14104.574} C_VEL
LIN {X 0,Y 349.887,Z 473.487,A -85,B 0,C 180,E1 -14105.842,E2 -14105.842} C_VEL
LIN {X 0,Y 347.94,Z 485.111,A -85,B 0,C 180,E1 -14107.276,E2 -14107.276} C_VEL
LIN {X 0,Y 346.112,Z 495.656,A -85,B 0,C 180,E1 -14108.825,E2 -14108.825} C_VEL
LIN {X 0,Y 344.405,Z 505.978,A -85,B 0,C 180,E1 -14110.635,E2 -14110.635} C_VEL
LIN {X 0,Y 342.61,Z 515.798,A -85,B 0,C 180,E1 -14112.697,E2 -14112.697} C_VEL
LIN {X 0,Y 341.321,Z 524.009,A -85,B 0,C 180,E1 -14114.78,E2 -14114.78} C_VEL
LIN {X 0,Y 340.375,Z 530.808,A -85,B 0,C 180,E1 -14116.873,E2 -14116.873} C_VEL
LIN {X 0,Y 339.606,Z 537.094,A -85,B 0,C 180,E1 -14119.266,E2 -14119.266} C_VEL
LIN {X 0,Y 339.278,Z 541.97,A -85,B 0,C 180,E1 -14121.663,E2 -14121.663} C_VEL
LIN {X 0,Y 339.128,Z 545.629,A -85,B 0,C 180,E1 -14124.119,E2 -14124.119} C_VEL
LIN {X 0,Y 339.092,Z 547.901,A -85,B 0,C 180,E1 -14126.436,E2 -14126.436} C_VEL
LIN {X 0,Y 339.179,Z 549.09,A -85,B 0,C 180,E1 -14128.813,E2 -14128.813} C_VEL
LIN {X 0,Y 339.179,Z 549.088,A -85,B 0,C 180,E1 -14131.188,E2 -14131.188} C_VEL
LIN {X 0,Y 339.096,Z 547.889,A -85,B 0,C 180,E1 -14133.565,E2 -14133.565} C_VEL
LIN {X 0,Y 339.206,Z 545.455,A -85,B 0,C 180,E1 -14136.007,E2 -14136.007} C_VEL
LIN {X 0,Y 339.28,Z 541.948,A -85,B 0,C 180,E1 -14138.338,E2 -14138.338} C_VEL
LIN {X 0,Y 339.607,Z 537.067,A -85,B 0,C 180,E1 -14140.735,E2 -14140.735} C_VEL
LIN {X 0,Y 340.38,Z 530.764,A -85,B 0,C 180,E1 -14143.128,E2 -14143.128} C_VEL
LIN {X 0,Y 341.482,Z 522.859,A -85,B 0,C 180,E1 -14145.519,E2 -14145.519} C_VEL
LIN {X 0,Y 342.795,Z 514.465,A -85,B 0,C 180,E1 -14147.603,E2 -14147.603} C_VEL
LIN {X 0,Y 344.633,Z 504.373,A -85,B 0,C 180,E1 -14149.663,E2 -14149.663} C_VEL
LIN {X 0,Y 346.363,Z 494.056,A -85,B 0,C 180,E1 -14151.423,E2 -14151.423} C_VEL
LIN {X 0,Y 348.461,Z 481.777,A -85,B 0,C 180,E1 -14153.16,E2 -14153.16} C_VEL
LIN {X 0,Y 350.742,Z 468.121,A -85,B 0,C 180,E1 -14154.727,E2 -14154.727} C_VEL
LIN {X 0,Y 352.834,Z 454.441,A -85,B 0,C 180,E1 -14155.99,E2 -14155.99} C_VEL
LIN {X 0,Y 353.579,Z 447.333,A -85,B 0,C 180,E1 -14156.562,E2 -14156.562} C_VEL
LIN {X 0,Y 351.719,Z 433.458,A -85,B 0,C 180,E1 -14157.752,E2 -14157.752} C_VEL
LIN {X 0,Y 348.503,Z 417.58,A -85,B 0,C 180,E1 -14158.947,E2 -14158.947} C_VEL
LIN {X 0,Y 344.124,Z 401.902,A -85,B 0,C 180,E1 -14159.986,E2 -14159.986} C_VEL
LIN {X 0,Y 341.16,Z 392.628,A -85,B 0,C 180,E1 -14160.527,E2 -14160.527} C_VEL
LIN {X 0,Y 341.127,Z 392.101,A -85,B 0,C 180,E1 -14160.571,E2 -14160.571} C_VEL
LIN {X 0,Y 341.881,Z 385.712,A -85,B 0,C 180,E1 -14164.687,E2 -14164.687} C_VEL
LIN {X 0,Y 342.422,Z 380.634,A -85,B 0,C 180,E1 -14168.006,E2 -14168.006} C_VEL
LIN {X 0,Y 343.115,Z 375.224,A -85,B 0,C 180,E1 -14171.718,E2 -14171.718} C_VEL
LIN {X 0,Y 342.915,Z 371.836,A -85,B 0,C 180,E1 -14174.174,E2 -14174.174} C_VEL
LIN {X 0,Y 342.191,Z 367.39,A -85,B 0,C 180,E1 -14177.679,E2 -14177.679} C_VEL
LIN {X 0,Y 341.483,Z 363.014,A -85,B 0,C 180,E1 -14181.451,E2 -14181.451} C_VEL
LIN {X 0,Y 340.784,Z 359.021,A -85,B 0,C 180,E1 -14185.223,E2 -14185.223} C_VEL
LIN {X 0,Y 340.725,Z 358.671,A -85,B 0,C 180,E1 -14185.596,E2 -14185.596} C_VEL
LIN {X 0,Y 340.7,Z 358.671,A -85,B 0,C 180,E1 -14188.956,E2 -14188.956} C_VEL
LIN {X 0,Y 340.806,Z 358.659,A -85,B 0,C 180,E1 -14193.02,E2 -14193.02} C_VEL
LIN {X 0,Y 340.759,Z 358.666,A -85,B 0,C 180,E1 -14195.639,E2 -14195.639} C_VEL
LIN {X 0,Y 340.759,Z 358.665,A -85,B 0,C 180,E1 -14199.475,E2 -14199.475} C_VEL
LIN {X 0,Y 340.861,Z 358.653,A -85,B 0,C 180,E1 -14201.985,E2 -14201.985} C_VEL
LIN {X 0,Y 340.872,Z 358.654,A -85,B 0,C 180,E1 -14205.705,E2 -14205.705} C_VEL
LIN {X 0,Y 340.874,Z 358.655,A -85,B 0,C 180,E1 -14209.306,E2 -14209.306} C_VEL
LIN {X 0,Y 341.079,Z 358.625,A -85,B 0,C 180,E1 -14212.898,E2 -14212.898} C_VEL
LIN {X 0,Y 341.173,Z 358.611,A -85,B 0,C 180,E1 -14217.639,E2 -14217.639} C_VEL
LIN {X 0,Y 341.298,Z 358.594,A -85,B 0,C 180,E1 -14220,E2 -14220} C_VEL
LIN {X 0,Y 341.173,Z 358.612,A -85,B 0,C 180,E1 -14222.361,E2 -14222.361} C_VEL
LIN {X 0,Y 341.08,Z 358.619,A -85,B 0,C 180,E1 -14227.102,E2 -14227.102} C_VEL
LIN {X 0,Y 340.875,Z 358.641,A -85,B 0,C 180,E1 -14230.694,E2 -14230.694} C_VEL
LIN {X 0,Y 340.866,Z 358.637,A -85,B 0,C 180,E1 -14234.325,E2 -14234.325} C_VEL
LIN {X 0,Y 340.84,Z 358.645,A -85,B 0,C 180,E1 -14238.466,E2 -14238.466} C_VEL
LIN {X 0,Y 340.724,Z 358.656,A -85,B 0,C 180,E1 -14241.843,E2 -14241.843} C_VEL
LIN {X 0,Y 340.775,Z 358.653,A -85,B 0,C 180,E1 -14245.664,E2 -14245.664} C_VEL
LIN {X 0,Y 340.731,Z 358.655,A -85,B 0,C 180,E1 -14248.321,E2 -14248.321} C_VEL
LIN {X 0,Y 340.701,Z 358.67,A -85,B 0,C 180,E1 -14251.045,E2 -14251.045} C_VEL
LIN {X 0,Y 340.721,Z 358.668,A -85,B 0,C 180,E1 -14255.279,E2 -14255.279} C_VEL
LIN {X 0,Y 340.713,Z 358.67,A -85,B 0,C 180,E1 -14258.386,E2 -14258.386} C_VEL
LIN {X 0,Y 340.702,Z 358.673,A -85,B 0,C 180,E1 -14262.045,E2 -14262.045} C_VEL
LIN {X 0,Y 340.648,Z 358.683,A -85,B 0,C 180,E1 -14266.228,E2 -14266.228} C_VEL
LIN {X 0,Y 340.585,Z 358.691,A -85,B 0,C 180,E1 -14268.675,E2 -14268.675} C_VEL
LIN {X 0,Y 340.468,Z 358.703,A -85,B 0,C 180,E1 -14270.214,E2 -14270.214} C_VEL
LIN {X 0,Y 340.368,Z 359.335,A -85,B 0,C 180,E1 -14271.724,E2 -14271.724} C_VEL
LIN {X 0,Y 340.274,Z 362.157,A -85,B 0,C 180,E1 -14275.706,E2 -14275.706} C_VEL
LIN {X 0,Y 340.132,Z 365.099,A -85,B 0,C 180,E1 -14279.446,E2 -14279.446} C_VEL
LIN {X 0,Y 341.171,Z 368.147,A -85,B 0,C 180,E1 -14279.637,E2 -14279.637} C_VEL
LIN {X 0,Y 346.762,Z 381.129,A -85,B 0,C 180,E1 -14280.634,E2 -14280.634} C_VEL
LIN {X 0,Y 351.727,Z 395.36,A -85,B 0,C 180,E1 -14281.813,E2 -14281.813} C_VEL
LIN {X 0,Y 355.525,Z 409.652,A -85,B 0,C 180,E1 -14283.111,E2 -14283.111} C_VEL
LIN {X 0,Y 355.418,Z 413.01,A -85,B 0,C 180,E1 -14283.372,E2 -14283.372} C_VEL
LIN {X 0,Y 353.635,Z 427.593,A -85,B 0,C 180,E1 -14284.547,E2 -14284.547} C_VEL
LIN {X 0,Y 351.84,Z 440.327,A -85,B 0,C 180,E1 -14285.827,E2 -14285.827} C_VEL
LIN {X 0,Y 349.88,Z 452.093,A -85,B 0,C 180,E1 -14287.252,E2 -14287.252} C_VEL
LIN {X 0,Y 347.832,Z 463.863,A -85,B 0,C 180,E1 -14288.983,E2 -14288.983} C_VEL
LIN {X 0,Y 346.056,Z 473.756,A -85,B 0,C 180,E1 -14290.73,E2 -14290.73} C_VEL
LIN {X 0,Y 344.254,Z 483.411,A -85,B 0,C 180,E1 -14292.781,E2 -14292.781} C_VEL
LIN {X 0,Y 342.759,Z 491.45,A -85,B 0,C 180,E1 -14294.845,E2 -14294.845} C_VEL
LIN {X 0,Y 341.614,Z 498.074,A -85,B 0,C 180,E1 -14296.92,E2 -14296.92} C_VEL
LIN {X 0,Y 340.651,Z 504.201,A -85,B 0,C 180,E1 -14299.299,E2 -14299.299} C_VEL
LIN {X 0,Y 339.974,Z 508.928,A -85,B 0,C 180,E1 -14301.679,E2 -14301.679} C_VEL
LIN {X 0,Y 339.55,Z 512.387,A -85,B 0,C 180,E1 -14304.059,E2 -14304.059} C_VEL
LIN {X 0,Y 339.3,Z 514.673,A -85,B 0,C 180,E1 -14306.437,E2 -14306.437} C_VEL
LIN {X 0,Y 339.272,Z 515.836,A -85,B 0,C 180,E1 -14308.813,E2 -14308.813} C_VEL
LIN {X 0,Y 339.273,Z 515.85,A -85,B 0,C 180,E1 -14311.186,E2 -14311.186} C_VEL
LIN {X 0,Y 339.299,Z 514.745,A -85,B 0,C 180,E1 -14313.562,E2 -14313.562} C_VEL
LIN {X 0,Y 339.549,Z 512.516,A -85,B 0,C 180,E1 -14315.94,E2 -14315.94} C_VEL
LIN {X 0,Y 339.963,Z 509.109,A -85,B 0,C 180,E1 -14318.32,E2 -14318.32} C_VEL
LIN {X 0,Y 340.621,Z 504.441,A -85,B 0,C 180,E1 -14320.701,E2 -14320.701} C_VEL
LIN {X 0,Y 341.571,Z 498.387,A -85,B 0,C 180,E1 -14323.081,E2 -14323.081} C_VEL
LIN {X 0,Y 342.789,Z 491.35,A -85,B 0,C 180,E1 -14325.29,E2 -14325.29} C_VEL
LIN {X 0,Y 344.425,Z 482.606,A -85,B 0,C 180,E1 -14327.516,E2 -14327.516} C_VEL
LIN {X 0,Y 346.299,Z 472.779,A -85,B 0,C 180,E1 -14329.564,E2 -14329.564} C_VEL
LIN {X 0,Y 348.087,Z 462.7,A -85,B 0,C 180,E1 -14331.31,E2 -14331.31} C_VEL
LIN {X 0,Y 350.138,Z 450.687,A -85,B 0,C 180,E1 -14333.041,E2 -14333.041} C_VEL
LIN {X 0,Y 352.148,Z 438.626,A -85,B 0,C 180,E1 -14334.463,E2 -14334.463} C_VEL
LIN {X 0,Y 353.758,Z 427.089,A -85,B 0,C 180,E1 -14335.6,E2 -14335.6} C_VEL
LIN {X 0,Y 355.462,Z 412.927,A -85,B 0,C 180,E1 -14336.737,E2 -14336.737} C_VEL
LIN {X 0,Y 355.654,Z 410.995,A -85,B 0,C 180,E1 -14336.877,E2 -14336.877} C_VEL
LIN {X 0,Y 354.7,Z 406.149,A -85,B 0,C 180,E1 -14337.318,E2 -14337.318} C_VEL
LIN {X 0,Y 350.772,Z 392.457,A -85,B 0,C 180,E1 -14338.54,E2 -14338.54} C_VEL
LIN {X 0,Y 345.656,Z 378.354,A -85,B 0,C 180,E1 -14339.692,E2 -14339.692} C_VEL
LIN {X 0,Y 340.244,Z 365.749,A -85,B 0,C 180,E1 -14340.636,E2 -14340.636} C_VEL
LIN {X 0,Y 340.099,Z 365.023,A -85,B 0,C 180,E1 -14340.683,E2 -14340.683} C_VEL
LIN {X 0,Y 340.276,Z 362.249,A -85,B 0,C 180,E1 -14344.294,E2 -14344.294} C_VEL
LIN {X 0,Y 340.386,Z 359.37,A -85,B 0,C 180,E1 -14348.317,E2 -14348.317} C_VEL
LIN {X 0,Y 340.494,Z 358.695,A -85,B 0,C 180,E1 -14350.208,E2 -14350.208} C_VEL
LIN {X 0,Y 340.641,Z 358.675,A -85,B 0,C 180,E1 -14353.143,E2 -14353.143} C_VEL
LIN {X 0,Y 339.963,Z 358.761,A -85,B 0,C 180,E1 -14354.129,E2 -14354.129} C_VEL
LIN {X 0,Y 337.117,Z 359.118,A -85,B 0,C 180,E1 -14355.733,E2 -14355.733} C_VEL
LIN {X 0,Y 334.716,Z 359.417,A -85,B 0,C 180,E1 -14357.032,E2 -14357.032} C_VEL
LIN {X 0,Y 333.691,Z 359.545,A -85,B 0,C 180,E1 -14358.037,E2 -14358.037} C_VEL
LIN {X 0,Y 333.609,Z 359.552,A -85,B 0,C 180,E1 -14358.377,E2 -14358.377} C_VEL
LIN {X 0,Y 333.651,Z 359.548,A -85,B 0,C 180,E1 -14361.201,E2 -14361.201} C_VEL
LIN {X 0,Y 333.675,Z 359.548,A -85,B 0,C 180,E1 -14363.861,E2 -14363.861} C_VEL
LIN {X 0,Y 333.644,Z 359.536,A -85,B 0,C 180,E1 -14367.412,E2 -14367.412} C_VEL
LIN {X 0,Y 333.71,Z 359.538,A -85,B 0,C 180,E1 -14371.028,E2 -14371.028} C_VEL
LIN {X 0,Y 333.734,Z 359.525,A -85,B 0,C 180,E1 -14373.753,E2 -14373.753} C_VEL
LIN {X 0,Y 333.717,Z 359.532,A -85,B 0,C 180,E1 -14377.914,E2 -14377.914} C_VEL
LIN {X 0,Y 333.791,Z 359.525,A -85,B 0,C 180,E1 -14381.589,E2 -14381.589} C_VEL
LIN {X 0,Y 333.806,Z 359.516,A -85,B 0,C 180,E1 -14385.576,E2 -14385.576} C_VEL
LIN {X 0,Y 333.836,Z 359.52,A -85,B 0,C 180,E1 -14389.078,E2 -14389.078} C_VEL
LIN {X 0,Y 334.024,Z 359.505,A -85,B 0,C 180,E1 -14392.747,E2 -14392.747} C_VEL
LIN {X 0,Y 333.81,Z 359.53,A -85,B 0,C 180,E1 -14395.169,E2 -14395.169} C_VEL
LIN {X 0,Y 334.105,Z 359.494,A -85,B 0,C 180,E1 -14397.589,E2 -14397.589} C_VEL
LIN {X 0,Y 334.264,Z 359.476,A -85,B 0,C 180,E1 -14400,E2 -14400} C_VEL
LIN {X 0,Y 334.106,Z 359.492,A -85,B 0,C 180,E1 -14402.411,E2 -14402.411} C_VEL
LIN {X 0,Y 334.023,Z 359.504,A -85,B 0,C 180,E1 -14407.252,E2 -14407.252} C_VEL
LIN {X 0,Y 333.832,Z 359.529,A -85,B 0,C 180,E1 -14410.922,E2 -14410.922} C_VEL
LIN {X 0,Y 333.806,Z 359.528,A -85,B 0,C 180,E1 -14414.634,E2 -14414.634} C_VEL
LIN {X 0,Y 333.794,Z 359.53,A -85,B 0,C 180,E1 -14418.655,E2 -14418.655} C_VEL
LIN {X 0,Y 333.69,Z 359.545,A -85,B 0,C 180,E1 -14422.278,E2 -14422.278} C_VEL
LIN {X 0,Y 333.733,Z 359.543,A -85,B 0,C 180,E1 -14426.246,E2 -14426.246} C_VEL
LIN {X 0,Y 333.709,Z 359.545,A -85,B 0,C 180,E1 -14428.972,E2 -14428.972} C_VEL
LIN {X 0,Y 333.643,Z 359.55,A -85,B 0,C 180,E1 -14432.588,E2 -14432.588} C_VEL
LIN {X 0,Y 333.683,Z 359.674,A -85,B 0,C 180,E1 -14433.927,E2 -14433.927} C_VEL
LIN {X 0,Y 334.319,Z 363.387,A -85,B 0,C 180,E1 -14437.563,E2 -14437.563} C_VEL
LIN {X 0,Y 334.959,Z 367.156,A -85,B 0,C 180,E1 -14440.946,E2 -14440.946} C_VEL
LIN {X 0,Y 335.697,Z 371.588,A -85,B 0,C 180,E1 -14444.619,E2 -14444.619} C_VEL
LIN {X 0,Y 336.058,Z 374.722,A -85,B 0,C 180,E1 -14447.051,E2 -14447.051} C_VEL
LIN {X 0,Y 335.997,Z 377.188,A -85,B 0,C 180,E1 -14448.851,E2 -14448.851} C_VEL
LIN {X 0,Y 335.299,Z 382.547,A -85,B 0,C 180,E1 -14452.566,E2 -14452.566} C_VEL
LIN {X 0,Y 334.676,Z 387.932,A -85,B 0,C 180,E1 -14456.188,E2 -14456.188} C_VEL
LIN {X 0,Y 334.163,Z 391.759,A -85,B 0,C 180,E1 -14458.716,E2 -14458.716} C_VEL
LIN {X 0,Y 335.104,Z 395.158,A -85,B 0,C 180,E1 -14458.917,E2 -14458.917} C_VEL
LIN {X 0,Y 339.478,Z 409.112,A -85,B 0,C 180,E1 -14459.821,E2 -14459.821} C_VEL
LIN {X 0,Y 342.964,Z 422.816,A -85,B 0,C 180,E1 -14460.826,E2 -14460.826} C_VEL
LIN {X 0,Y 345.539,Z 436.711,A -85,B 0,C 180,E1 -14461.952,E2 -14461.952} C_VEL
LIN {X 0,Y 347.038,Z 448.412,A -85,B 0,C 180,E1 -14463.007,E2 -14463.007} C_VEL
LIN {X 0,Y 345.263,Z 462.187,A -85,B 0,C 180,E1 -14464.209,E2 -14464.209} C_VEL
LIN {X 0,Y 342.966,Z 475.657,A -85,B 0,C 180,E1 -14465.645,E2 -14465.645} C_VEL
LIN {X 0,Y 340.685,Z 487.934,A -85,B 0,C 180,E1 -14467.245,E2 -14467.245} C_VEL
LIN {X 0,Y 338.647,Z 499.3,A -85,B 0,C 180,E1 -14469.05,E2 -14469.05} C_VEL
LIN {X 0,Y 337.038,Z 508.627,A -85,B 0,C 180,E1 -14470.827,E2 -14470.827} C_VEL
LIN {X 0,Y 335.312,Z 517.941,A -85,B 0,C 180,E1 -14472.937,E2 -14472.937} C_VEL
LIN {X 0,Y 333.915,Z 526.726,A -85,B 0,C 180,E1 -14475.371,E2 -14475.371} C_VEL
LIN {X 0,Y 332.982,Z 533.79,A -85,B 0,C 180,E1 -14477.816,E2 -14477.816} C_VEL
LIN {X 0,Y 332.339,Z 539.35,A -85,B 0,C 180,E1 -14480.261,E2 -14480.261} C_VEL
LIN {X 0,Y 332.136,Z 543.568,A -85,B 0,C 180,E1 -14482.707,E2 -14482.707} C_VEL
LIN {X 0,Y 332.016,Z 546.525,A -85,B 0,C 180,E1 -14485.143,E2 -14485.143} C_VEL
LIN {X 0,Y 332.001,Z 548.29,A -85,B 0,C 180,E1 -14487.574,E2 -14487.574} C_VEL
LIN {X 0,Y 332.13,Z 548.9,A -85,B 0,C 180,E1 -14490.001,E2 -14490.001} C_VEL
LIN {X 0,Y 332.002,Z 548.283,A -85,B 0,C 180,E1 -14492.427,E2 -14492.427} C_VEL
LIN {X 0,Y 332.043,Z 546.508,A -85,B 0,C 180,E1 -14494.857,E2 -14494.857} C_VEL
LIN {X 0,Y 332.141,Z 543.545,A -85,B 0,C 180,E1 -14497.294,E2 -14497.294} C_VEL
LIN {X 0,Y 332.34,Z 539.325,A -85,B 0,C 180,E1 -14499.74,E2 -14499.74} C_VEL
LIN {X 0,Y 332.985,Z 533.753,A -85,B 0,C 180,E1 -14502.185,E2 -14502.185} C_VEL
LIN {X 0,Y 333.916,Z 526.671,A -85,B 0,C 180,E1 -14504.63,E2 -14504.63} C_VEL
LIN {X 0,Y 335.313,Z 517.877,A -85,B 0,C 180,E1 -14507.064,E2 -14507.064} C_VEL
LIN {X 0,Y 337.007,Z 508.551,A -85,B 0,C 180,E1 -14509.175,E2 -14509.175} C_VEL
LIN {X 0,Y 338.782,Z 498.858,A -85,B 0,C 180,E1 -14511.01,E2 -14511.01} C_VEL
LIN {X 0,Y 340.798,Z 487.843,A -85,B 0,C 180,E1 -14512.748,E2 -14512.748} C_VEL
LIN {X 0,Y 342.964,Z 475.542,A -85,B 0,C 180,E1 -14514.356,E2 -14514.356} C_VEL
LIN {X 0,Y 345.266,Z 462.032,A -85,B 0,C 180,E1 -14515.792,E2 -14515.792} C_VEL
LIN {X 0,Y 347.003,Z 448.378,A -85,B 0,C 180,E1 -14516.982,E2 -14516.982} C_VEL
LIN {X 0,Y 345.131,Z 434.054,A -85,B 0,C 180,E1 -14518.258,E2 -14518.258} C_VEL
LIN {X 0,Y 342.095,Z 418.932,A -85,B 0,C 180,E1 -14519.449,E2 -14519.449} C_VEL
LIN {X 0,Y 337.844,Z 403.512,A -85,B 0,C 180,E1 -14520.529,E2 -14520.529} C_VEL
LIN {X 0,Y 334.233,Z 392.643,A -85,B 0,C 180,E1 -14521.219,E2 -14521.219} C_VEL
LIN {X 0,Y 334.128,Z 391.763,A -85,B 0,C 180,E1 -14521.266,E2 -14521.266} C_VEL
LIN {X 0,Y 334.89,Z 386.021,A -85,B 0,C 180,E1 -14525.07,E2 -14525.07} C_VEL
LIN {X 0,Y 335.541,Z 380.298,A -85,B 0,C 180,E1 -14528.93,E2 -14528.93} C_VEL
LIN {X 0,Y 336.12,Z 375.964,A -85,B 0,C 180,E1 -14531.998,E2 -14531.998} C_VEL
LIN {X 0,Y 335.839,Z 372.451,A -85,B 0,C 180,E1 -14534.642,E2 -14534.642} C_VEL
LIN {X 0,Y 335.183,Z 368.526,A -85,B 0,C 180,E1 -14537.859,E2 -14537.859} C_VEL
LIN {X 0,Y 334.601,Z 364.867,A -85,B 0,C 180,E1 -14541.001,E2 -14541.001} C_VEL
LIN {X 0,Y 334.075,Z 361.8,A -85,B 0,C 180,E1 -14543.911,E2 -14543.911} C_VEL
LIN {X 0,Y 333.668,Z 359.55,A -85,B 0,C 180,E1 -14546.253,E2 -14546.253} C_VEL
LIN {X 0,Y 333.697,Z 359.543,A -85,B 0,C 180,E1 -14549.713,E2 -14549.713} C_VEL
LIN {X 0,Y 333.742,Z 359.541,A -85,B 0,C 180,E1 -14552.401,E2 -14552.401} C_VEL
LIN {X 0,Y 333.729,Z 359.541,A -85,B 0,C 180,E1 -14555.091,E2 -14555.091} C_VEL
LIN {X 0,Y 333.69,Z 359.545,A -85,B 0,C 180,E1 -14559.02,E2 -14559.02} C_VEL
LIN {X 0,Y 333.797,Z 359.533,A -85,B 0,C 180,E1 -14561.59,E2 -14561.59} C_VEL
LIN {X 0,Y 333.811,Z 359.533,A -85,B 0,C 180,E1 -14565.577,E2 -14565.577} C_VEL
LIN {X 0,Y 333.837,Z 359.531,A -85,B 0,C 180,E1 -14569.078,E2 -14569.078} C_VEL
LIN {X 0,Y 334.029,Z 359.504,A -85,B 0,C 180,E1 -14572.748,E2 -14572.748} C_VEL
LIN {X 0,Y 333.814,Z 359.532,A -85,B 0,C 180,E1 -14575.169,E2 -14575.169} C_VEL
LIN {X 0,Y 334.11,Z 359.491,A -85,B 0,C 180,E1 -14577.589,E2 -14577.589} C_VEL
LIN {X 0,Y 334.249,Z 359.472,A -85,B 0,C 180,E1 -14580,E2 -14580} C_VEL
LIN {X 0,Y 334.11,Z 359.492,A -85,B 0,C 180,E1 -14582.411,E2 -14582.411} C_VEL
LIN {X 0,Y 334.029,Z 359.498,A -85,B 0,C 180,E1 -14587.253,E2 -14587.253} C_VEL
LIN {X 0,Y 333.837,Z 359.516,A -85,B 0,C 180,E1 -14590.922,E2 -14590.922} C_VEL
LIN {X 0,Y 333.812,Z 359.518,A -85,B 0,C 180,E1 -14594.634,E2 -14594.634} C_VEL
LIN {X 0,Y 333.799,Z 359.521,A -85,B 0,C 180,E1 -14598.655,E2 -14598.655} C_VEL
LIN {X 0,Y 333.663,Z 359.539,A -85,B 0,C 180,E1 -14602.28,E2 -14602.28} C_VEL
LIN {X 0,Y 333.738,Z 359.525,A -85,B 0,C 180,E1 -14606.246,E2 -14606.246} C_VEL
LIN {X 0,Y 333.693,Z 359.537,A -85,B 0,C 180,E1 -14608.974,E2 -14608.974} C_VEL
LIN {X 0,Y 333.646,Z 359.538,A -85,B 0,C 180,E1 -14612.587,E2 -14612.587} C_VEL
LIN {X 0,Y 333.68,Z 359.547,A -85,B 0,C 180,E1 -14616.139,E2 -14616.139} C_VEL
LIN {X 0,Y 333.65,Z 359.55,A -85,B 0,C 180,E1 -14619.192,E2 -14619.192} C_VEL
LIN {X 0,Y 333.636,Z 359.555,A -85,B 0,C 180,E1 -14622.5,E2 -14622.5} C_VEL
LIN {X 0,Y 333.593,Z 359.561,A -85,B 0,C 180,E1 -14625.954,E2 -14625.954} C_VEL
LIN {X 0,Y 333.508,Z 359.571,A -85,B 0,C 180,E1 -14629.211,E2 -14629.211} C_VEL
LIN {X 0,Y 333.357,Z 359.681,A -85,B 0,C 180,E1 -14630.766,E2 -14630.766} C_VEL
LIN {X 0,Y 333.257,Z 361.78,A -85,B 0,C 180,E1 -14633.808,E2 -14633.808} C_VEL
LIN {X 0,Y 333.171,Z 363.914,A -85,B 0,C 180,E1 -14636.739,E2 -14636.739} C_VEL
LIN {X 0,Y 333.126,Z 365.461,A -85,B 0,C 180,E1 -14638.73,E2 -14638.73} C_VEL
LIN {X 0,Y 334.123,Z 368.459,A -85,B 0,C 180,E1 -14638.923,E2 -14638.923} C_VEL
LIN {X 0,Y 339.426,Z 380.46,A -85,B 0,C 180,E1 -14639.885,E2 -14639.885} C_VEL
LIN {X 0,Y 344.333,Z 394.127,A -85,B 0,C 180,E1 -14641.057,E2 -14641.057} C_VEL
LIN {X 0,Y 347.848,Z 406.329,A -85,B 0,C 180,E1 -14642.191,E2 -14642.191} C_VEL
LIN {X 0,Y 349.207,Z 412.447,A -85,B 0,C 180,E1 -14642.785,E2 -14642.785} C_VEL
LIN {X 0,Y 347.48,Z 426.372,A -85,B 0,C 180,E1 -14643.902,E2 -14643.902} C_VEL
LIN {X 0,Y 345.796,Z 438.113,A -85,B 0,C 180,E1 -14645.056,E2 -14645.056} C_VEL
LIN {X 0,Y 343.721,Z 450.31,A -85,B 0,C 180,E1 -14646.502,E2 -14646.502} C_VEL
LIN {X 0,Y 341.581,Z 462.445,A -85,B 0,C 180,E1 -14648.262,E2 -14648.262} C_VEL
LIN {X 0,Y 339.682,Z 472.585,A -85,B 0,C 180,E1 -14650.038,E2 -14650.038} C_VEL
LIN {X 0,Y 337.718,Z 482.502,A -85,B 0,C 180,E1 -14652.124,E2 -14652.124} C_VEL
LIN {X 0,Y 335.931,Z 491.424,A -85,B 0,C 180,E1 -14654.417,E2 -14654.417} C_VEL
LIN {X 0,Y 334.701,Z 498.424,A -85,B 0,C 180,E1 -14656.645,E2 -14656.645} C_VEL
LIN {X 0,Y 333.674,Z 504.55,A -85,B 0,C 180,E1 -14659.072,E2 -14659.072} C_VEL
LIN {X 0,Y 332.931,Z 509.278,A -85,B 0,C 180,E1 -14661.502,E2 -14661.502} C_VEL
LIN {X 0,Y 332.497,Z 512.735,A -85,B 0,C 180,E1 -14663.933,E2 -14663.933} C_VEL
LIN {X 0,Y 332.222,Z 515.021,A -85,B 0,C 180,E1 -14666.361,E2 -14666.361} C_VEL
LIN {X 0,Y 332.181,Z 516.183,A -85,B 0,C 180,E1 -14668.787,E2 -14668.787} C_VEL
LIN {X 0,Y 332.182,Z 516.197,A -85,B 0,C 180,E1 -14671.212,E2 -14671.212} C_VEL
LIN {X 0,Y 332.221,Z 515.093,A -85,B 0,C 180,E1 -14673.638,E2 -14673.638} C_VEL
LIN {X 0,Y 332.496,Z 512.863,A -85,B 0,C 180,E1 -14676.066,E2 -14676.066} C_VEL
LIN {X 0,Y 332.917,Z 509.457,A -85,B 0,C 180,E1 -14678.497,E2 -14678.497} C_VEL
LIN {X 0,Y 333.627,Z 504.789,A -85,B 0,C 180,E1 -14680.928,E2 -14680.928} C_VEL
LIN {X 0,Y 334.654,Z 498.734,A -85,B 0,C 180,E1 -14683.356,E2 -14683.356} C_VEL
LIN {X 0,Y 335.855,Z 492.039,A -85,B 0,C 180,E1 -14685.508,E2 -14685.508} C_VEL
LIN {X 0,Y 337.648,Z 482.952,A -85,B 0,C 180,E1 -14687.879,E2 -14687.879} C_VEL
LIN {X 0,Y 339.6,Z 473.125,A -85,B 0,C 180,E1 -14689.966,E2 -14689.966} C_VEL
LIN {X 0,Y 341.48,Z 463.045,A -85,B 0,C 180,E1 -14691.743,E2 -14691.743} C_VEL
LIN {X 0,Y 343.615,Z 451.031,A -85,B 0,C 180,E1 -14693.505,E2 -14693.505} C_VEL
LIN {X 0,Y 345.701,Z 438.969,A -85,B 0,C 180,E1 -14694.95,E2 -14694.95} C_VEL
LIN {X 0,Y 347.386,Z 427.431,A -85,B 0,C 180,E1 -14696.105,E2 -14696.105} C_VEL
LIN {X 0,Y 349.132,Z 413.268,A -85,B 0,C 180,E1 -14697.262,E2 -14697.262} C_VEL
LIN {X 0,Y 349.108,Z 411.2,A -85,B 0,C 180,E1 -14697.435,E2 -14697.435} C_VEL
LIN {X 0,Y 345.489,Z 397.73,A -85,B 0,C 180,E1 -14698.721,E2 -14698.721} C_VEL
LIN {X 0,Y 340.828,Z 384.112,A -85,B 0,C 180,E1 -14699.915,E2 -14699.915} C_VEL
LIN {X 0,Y 334.571,Z 369.146,A -85,B 0,C 180,E1 -14701.122,E2 -14701.122} C_VEL
LIN {X 0,Y 333.215,Z 366.097,A -85,B 0,C 180,E1 -14701.355,E2 -14701.355} C_VEL
LIN {X 0,Y 333.099,Z 365.373,A -85,B 0,C 180,E1 -14701.433,E2 -14701.433} C_VEL
LIN {X 0,Y 333.235,Z 362.907,A -85,B 0,C 180,E1 -14704.71,E2 -14704.71} C_VEL
LIN {X 0,Y 333.317,Z 360.808,A -85,B 0,C 180,E1 -14707.695,E2 -14707.695} C_VEL
LIN {X 0,Y 333.359,Z 359.772,A -85,B 0,C 180,E1 -14709.232,E2 -14709.232} C_VEL
LIN {X 0,Y 333.597,Z 359.551,A -85,B 0,C 180,E1 -14712.388,E2 -14712.388} C_VEL
LIN {X 0,Y 333.594,Z 359.558,A -85,B 0,C 180,E1 -14715.954,E2 -14715.954} C_VEL
LIN {X 0,Y 333.609,Z 359.552,A -85,B 0,C 180,E1 -14718.377,E2 -14718.377} C_VEL
LIN {X 0,Y 332.951,Z 359.638,A -85,B 0,C 180,E1 -14719.385,E2 -14719.385} C_VEL
LIN {X 0,Y 330.115,Z 359.989,A -85,B 0,C 180,E1 -14721.025,E2 -14721.025} C_VEL
LIN {X 0,Y 327.708,Z 360.291,A -85,B 0,C 180,E1 -14722.353,E2 -14722.353} C_VEL
LIN {X 0,Y 326.675,Z 360.417,A -85,B 0,C 180,E1 -14723.381,E2 -14723.381} C_VEL
LIN {X 0,Y 326.591,Z 360.425,A -85,B 0,C 180,E1 -14723.729,E2 -14723.729} C_VEL
LIN {X 0,Y 326.608,Z 360.413,A -85,B 0,C 180,E1 -14727.455,E2 -14727.455} C_VEL
LIN {X 0,Y 326.659,Z 360.419,A -85,B 0,C 180,E1 -14730.341,E2 -14730.341} C_VEL
LIN {X 0,Y 326.688,Z 360.408,A -85,B 0,C 180,E1 -14734.516,E2 -14734.516} C_VEL
LIN {X 0,Y 326.643,Z 360.404,A -85,B 0,C 180,E1 -14738.545,E2 -14738.545} C_VEL
LIN {X 0,Y 326.742,Z 360.4,A -85,B 0,C 180,E1 -14741.177,E2 -14741.177} C_VEL
LIN {X 0,Y 326.761,Z 360.394,A -85,B 0,C 180,E1 -14745.433,E2 -14745.433} C_VEL
LIN {X 0,Y 326.771,Z 360.399,A -85,B 0,C 180,E1 -14748.839,E2 -14748.839} C_VEL
LIN {X 0,Y 326.977,Z 360.382,A -85,B 0,C 180,E1 -14752.59,E2 -14752.59} C_VEL
LIN {X 0,Y 326.777,Z 360.406,A -85,B 0,C 180,E1 -14755.065,E2 -14755.065} C_VEL
LIN {X 0,Y 327.046,Z 360.373,A -85,B 0,C 180,E1 -14757.537,E2 -14757.537} C_VEL
LIN {X 0,Y 327.215,Z 360.354,A -85,B 0,C 180,E1 -14760,E2 -14760} C_VEL
LIN {X 0,Y 327.046,Z 360.371,A -85,B 0,C 180,E1 -14762.463,E2 -14762.463} C_VEL
LIN {X 0,Y 326.994,Z 360.38,A -85,B 0,C 180,E1 -14766.169,E2 -14766.169} C_VEL
LIN {X 0,Y 326.912,Z 360.388,A -85,B 0,C 180,E1 -14768.655,E2 -14768.655} C_VEL
LIN {X 0,Y 326.732,Z 360.407,A -85,B 0,C 180,E1 -14772.421,E2 -14772.421} C_VEL
LIN {X 0,Y 326.751,Z 360.407,A -85,B 0,C 180,E1 -14774.957,E2 -14774.957} C_VEL
LIN {X 0,Y 326.731,Z 360.41,A -85,B 0,C 180,E1 -14778.839,E2 -14778.839} C_VEL
LIN {X 0,Y 326.618,Z 360.427,A -85,B 0,C 180,E1 -14782.787,E2 -14782.787} C_VEL
LIN {X 0,Y 326.687,Z 360.419,A -85,B 0,C 180,E1 -14785.484,E2 -14785.484} C_VEL
LIN {X 0,Y 326.658,Z 360.423,A -85,B 0,C 180,E1 -14789.659,E2 -14789.659} C_VEL
LIN {X 0,Y 326.626,Z 360.516,A -85,B 0,C 180,E1 -14793.271,E2 -14793.271} C_VEL
LIN {X 0,Y 327.293,Z 364.144,A -85,B 0,C 180,E1 -14796.959,E2 -14796.959} C_VEL
LIN {X 0,Y 327.791,Z 367.462,A -85,B 0,C 180,E1 -14800.032,E2 -14800.032} C_VEL
LIN {X 0,Y 328.436,Z 371.234,A -85,B 0,C 180,E1 -14803.32,E2 -14803.32} C_VEL
LIN {X 0,Y 328.824,Z 373.444,A -85,B 0,C 180,E1 -14805.146,E2 -14805.146} C_VEL
LIN {X 0,Y 329.044,Z 375.657,A -85,B 0,C 180,E1 -14806.884,E2 -14806.884} C_VEL
LIN {X 0,Y 328.878,Z 378.938,A -85,B 0,C 180,E1 -14809.325,E2 -14809.325} C_VEL
LIN {X 0,Y 328.154,Z 384.348,A -85,B 0,C 180,E1 -14813.155,E2 -14813.155} C_VEL
LIN {X 0,Y 327.452,Z 389.683,A -85,B 0,C 180,E1 -14816.829,E2 -14816.829} C_VEL
LIN {X 0,Y 327.24,Z 391.445,A -85,B 0,C 180,E1 -14817.993,E2 -14817.993} C_VEL
LIN {X 0,Y 328.187,Z 394.807,A -85,B 0,C 180,E1 -14818.187,E2 -14818.187} C_VEL
LIN {X 0,Y 332.728,Z 408.924,A -85,B 0,C 180,E1 -14819.15,E2 -14819.15} C_VEL
LIN {X 0,Y 336.419,Z 423.438,A -85,B 0,C 180,E1 -14820.256,E2 -14820.256} C_VEL
LIN {X 0,Y 338.988,Z 437.346,A -85,B 0,C 180,E1 -14821.434,E2 -14821.434} C_VEL
LIN {X 0,Y 340.467,Z 449.482,A -85,B 0,C 180,E1 -14822.575,E2 -14822.575} C_VEL
LIN {X 0,Y 338.859,Z 461.842,A -85,B 0,C 180,E1 -14823.685,E2 -14823.685} C_VEL
LIN {X 0,Y 336.655,Z 474.091,A -85,B 0,C 180,E1 -14824.993,E2 -14824.993} C_VEL
LIN {X 0,Y 334.352,Z 486.568,A -85,B 0,C 180,E1 -14826.626,E2 -14826.626} C_VEL
LIN {X 0,Y 332.38,Z 497.045,A -85,B 0,C 180,E1 -14828.284,E2 -14828.284} C_VEL
LIN {X 0,Y 330.589,Z 506.778,A -85,B 0,C 180,E1 -14830.115,E2 -14830.115} C_VEL
LIN {X 0,Y 328.678,Z 516.344,A -85,B 0,C 180,E1 -14832.26,E2 -14832.26} C_VEL
LIN {X 0,Y 327.311,Z 524.331,A -85,B 0,C 180,E1 -14834.432,E2 -14834.432} C_VEL
LIN {X 0,Y 326.153,Z 531.799,A -85,B 0,C 180,E1 -14836.924,E2 -14836.924} C_VEL
LIN {X 0,Y 325.377,Z 537.732,A -85,B 0,C 180,E1 -14839.421,E2 -14839.421} C_VEL
LIN {X 0,Y 325.126,Z 541.27,A -85,B 0,C 180,E1 -14841.297,E2 -14841.297} C_VEL
LIN {X 0,Y 324.954,Z 544.849,A -85,B 0,C 180,E1 -14843.793,E2 -14843.793} C_VEL
LIN {X 0,Y 324.943,Z 547.207,A -85,B 0,C 180,E1 -14846.28,E2 -14846.28} C_VEL
LIN {X 0,Y 324.986,Z 548.394,A -85,B 0,C 180,E1 -14848.761,E2 -14848.761} C_VEL
LIN {X 0,Y 325.038,Z 548.553,A -85,B 0,C 180,E1 -14850.001,E2 -14850.001} C_VEL
LIN {X 0,Y 324.916,Z 547.935,A -85,B 0,C 180,E1 -14852.48,E2 -14852.48} C_VEL
LIN {X 0,Y 324.953,Z 546.159,A -85,B 0,C 180,E1 -14854.963,E2 -14854.963} C_VEL
LIN {X 0,Y 325.044,Z 543.194,A -85,B 0,C 180,E1 -14857.455,E2 -14857.455} C_VEL
LIN {X 0,Y 325.295,Z 538.974,A -85,B 0,C 180,E1 -14859.954,E2 -14859.954} C_VEL
LIN {X 0,Y 325.963,Z 533.399,A -85,B 0,C 180,E1 -14862.452,E2 -14862.452} C_VEL
LIN {X 0,Y 326.983,Z 526.318,A -85,B 0,C 180,E1 -14864.947,E2 -14864.947} C_VEL
LIN {X 0,Y 328.444,Z 517.522,A -85,B 0,C 180,E1 -14867.432,E2 -14867.432} C_VEL
LIN {X 0,Y 330.248,Z 508.198,A -85,B 0,C 180,E1 -14869.584,E2 -14869.584} C_VEL
LIN {X 0,Y 331.953,Z 499.23,A -85,B 0,C 180,E1 -14871.322,E2 -14871.322} C_VEL
LIN {X 0,Y 333.773,Z 489.453,A -85,B 0,C 180,E1 -14872.926,E2 -14872.926} C_VEL
LIN {X 0,Y 336.02,Z 477.551,A -85,B 0,C 180,E1 -14874.564,E2 -14874.564} C_VEL
LIN {X 0,Y 338.351,Z 464.547,A -85,B 0,C 180,E1 -14876.028,E2 -14876.028} C_VEL
LIN {X 0,Y 340.293,Z 451.555,A -85,B 0,C 180,E1 -14877.228,E2 -14877.228} C_VEL
LIN {X 0,Y 340.262,Z 447.579,A -85,B 0,C 180,E1 -14877.601,E2 -14877.601} C_VEL
LIN {X 0,Y 338.612,Z 435.357,A -85,B 0,C 180,E1 -14878.728,E2 -14878.728} C_VEL
LIN {X 0,Y 335.826,Z 420.906,A -85,B 0,C 180,E1 -14879.923,E2 -14879.923} C_VEL
LIN {X 0,Y 331.93,Z 406.146,A -85,B 0,C 180,E1 -14881.018,E2 -14881.018} C_VEL
LIN {X 0,Y 327.276,Z 392.026,A -85,B 0,C 180,E1 -14881.965,E2 -14881.965} C_VEL
LIN {X 0,Y 327.212,Z 391.347,A -85,B 0,C 180,E1 -14882.033,E2 -14882.033} C_VEL
LIN {X 0,Y 327.896,Z 386.466,A -85,B 0,C 180,E1 -14885.36,E2 -14885.36} C_VEL
LIN {X 0,Y 328.397,Z 382.115,A -85,B 0,C 180,E1 -14888.362,E2 -14888.362} C_VEL
LIN {X 0,Y 329.027,Z 377.583,A -85,B 0,C 180,E1 -14891.617,E2 -14891.617} C_VEL
LIN {X 0,Y 329.002,Z 375.226,A -85,B 0,C 180,E1 -14893.424,E2 -14893.424} C_VEL
LIN {X 0,Y 328.758,Z 373.036,A -85,B 0,C 180,E1 -14895.134,E2 -14895.134} C_VEL
LIN {X 0,Y 328.061,Z 368.972,A -85,B 0,C 180,E1 -14898.574,E2 -14898.574} C_VEL
LIN {X 0,Y 327.509,Z 365.686,A -85,B 0,C 180,E1 -14901.515,E2 -14901.515} C_VEL
LIN {X 0,Y 326.964,Z 362.38,A -85,B 0,C 180,E1 -14904.766,E2 -14904.766} C_VEL
LIN {X 0,Y 326.601,Z 360.431,A -85,B 0,C 180,E1 -14906.875,E2 -14906.875} C_VEL
LIN {X 0,Y 326.65,Z 360.423,A -85,B 0,C 180,E1 -14910.34,E2 -14910.34} C_VEL
LIN {X 0,Y 326.693,Z 360.418,A -85,B 0,C 180,E1 -14914.517,E2 -14914.517} C_VEL
LIN {X 0,Y 326.652,Z 360.423,A -85,B 0,C 180,E1 -14918.546,E2 -14918.546} C_VEL
LIN {X 0,Y 326.747,Z 360.41,A -85,B 0,C 180,E1 -14921.178,E2 -14921.178} C_VEL
LIN {X 0,Y 326.766,Z 360.41,A -85,B 0,C 180,E1 -14925.433,E2 -14925.433} C_VEL
LIN {X 0,Y 326.773,Z 360.41,A -85,B 0,C 180,E1 -14928.839,E2 -14928.839} C_VEL
LIN {X 0,Y 326.983,Z 360.382,A -85,B 0,C 180,E1 -14932.591,E2 -14932.591} C_VEL
LIN {X 0,Y 326.781,Z 360.407,A -85,B 0,C 180,E1 -14935.065,E2 -14935.065} C_VEL
LIN {X 0,Y 327.051,Z 360.37,A -85,B 0,C 180,E1 -14937.537,E2 -14937.537} C_VEL
LIN {X 0,Y 327.2,Z 360.35,A -85,B 0,C 180,E1 -14940,E2 -14940} C_VEL
LIN {X 0,Y 327.051,Z 360.371,A -85,B 0,C 180,E1 -14942.463,E2 -14942.463} C_VEL
LIN {X 0,Y 326.975,Z 360.375,A -85,B 0,C 180,E1 -14946.647,E2 -14946.647} C_VEL
LIN {X 0,Y 326.817,Z 360.399,A -85,B 0,C 180,E1 -14949.906,E2 -14949.906} C_VEL
LIN {X 0,Y 326.762,Z 360.382,A -85,B 0,C 180,E1 -14953.685,E2 -14953.685} C_VEL
LIN {X 0,Y 326.703,Z 360.413,A -85,B 0,C 180,E1 -14957.528,E2 -14957.528} C_VEL
LIN {X 0,Y 326.662,Z 360.393,A -85,B 0,C 180,E1 -14960.135,E2 -14960.135} C_VEL
LIN {X 0,Y 326.653,Z 360.422,A -85,B 0,C 180,E1 -14964.129,E2 -14964.129} C_VEL
LIN {X 0,Y 326.686,Z 360.397,A -85,B 0,C 180,E1 -14966.858,E2 -14966.858} C_VEL
LIN {X 0,Y 326.637,Z 360.423,A -85,B 0,C 180,E1 -14970.61,E2 -14970.61} C_VEL
LIN {X 0,Y 326.61,Z 360.412,A -85,B 0,C 180,E1 -14974.019,E2 -14974.019} C_VEL
LIN {X 0,Y 326.631,Z 360.424,A -85,B 0,C 180,E1 -14977.239,E2 -14977.239} C_VEL
LIN {X 0,Y 326.58,Z 360.431,A -85,B 0,C 180,E1 -14981.131,E2 -14981.131} C_VEL
LIN {X 0,Y 326.528,Z 360.44,A -85,B 0,C 180,E1 -14984.742,E2 -14984.742} C_VEL
LIN {X 0,Y 326.515,Z 360.443,A -85,B 0,C 180,E1 -14988.144,E2 -14988.144} C_VEL
LIN {X 0,Y 326.341,Z 360.742,A -85,B 0,C 180,E1 -14990.831,E2 -14990.831} C_VEL
LIN {X 0,Y 326.208,Z 363.566,A -85,B 0,C 180,E1 -14994.954,E2 -14994.954} C_VEL
LIN {X 0,Y 326.105,Z 365.797,A -85,B 0,C 180,E1 -14997.952,E2 -14997.952} C_VEL
LIN {X 0,Y 327.254,Z 369.025,A -85,B 0,C 180,E1 -14998.2,E2 -14998.2} C_VEL
LIN {X 0,Y 332.631,Z 381.048,A -85,B 0,C 180,E1 -14999.212,E2 -14999.212} C_VEL
LIN {X 0,Y 337.466,Z 394.311,A -85,B 0,C 180,E1 -15000.398,E2 -15000.398} C_VEL
LIN {X 0,Y 340.983,Z 406.107,A -85,B 0,C 180,E1 -15001.535,E2 -15001.535} C_VEL
LIN {X 0,Y 342.786,Z 413.895,A -85,B 0,C 180,E1 -15002.323,E2 -15002.323} C_VEL
LIN {X 0,Y 340.891,Z 428.298,A -85,B 0,C 180,E1 -15003.523,E2 -15003.523} C_VEL
LIN {X 0,Y 338.957,Z 441.031,A -85,B 0,C 180,E1 -15004.846,E2 -15004.846} C_VEL
LIN {X 0,Y 336.812,Z 452.797,A -85,B 0,C 180,E1 -15006.317,E2 -15006.317} C_VEL
LIN {X 0,Y 334.617,Z 464.565,A -85,B 0,C 180,E1 -15008.111,E2 -15008.111} C_VEL
LIN {X 0,Y 332.668,Z 474.458,A -85,B 0,C 180,E1 -15009.921,E2 -15009.921} C_VEL
LIN {X 0,Y 330.675,Z 484.113,A -85,B 0,C 180,E1 -15012.05,E2 -15012.05} C_VEL
LIN {X 0,Y 329.005,Z 492.111,A -85,B 0,C 180,E1 -15014.181,E2 -15014.181} C_VEL
LIN {X 0,Y 327.796,Z 498.773,A -85,B 0,C 180,E1 -15016.358,E2 -15016.358} C_VEL
LIN {X 0,Y 326.684,Z 504.901,A -85,B 0,C 180,E1 -15018.835,E2 -15018.835} C_VEL
LIN {X 0,Y 325.893,Z 509.627,A -85,B 0,C 180,E1 -15021.317,E2 -15021.317} C_VEL
LIN {X 0,Y 325.448,Z 513.083,A -85,B 0,C 180,E1 -15023.801,E2 -15023.801} C_VEL
LIN {X 0,Y 325.148,Z 515.369,A -85,B 0,C 180,E1 -15026.282,E2 -15026.282} C_VEL
LIN {X 0,Y 325.09,Z 516.531,A -85,B 0,C 180,E1 -15028.761,E2 -15028.761} C_VEL
LIN {X 0,Y 325.09,Z 516.545,A -85,B 0,C 180,E1 -15031.238,E2 -15031.238} C_VEL
LIN {X 0,Y 325.147,Z 515.44,A -85,B 0,C 180,E1 -15033.717,E2 -15033.717} C_VEL
LIN {X 0,Y 325.448,Z 513.209,A -85,B 0,C 180,E1 -15036.198,E2 -15036.198} C_VEL
LIN {X 0,Y 325.879,Z 509.805,A -85,B 0,C 180,E1 -15038.682,E2 -15038.682} C_VEL
LIN {X 0,Y 326.625,Z 505.137,A -85,B 0,C 180,E1 -15041.165,E2 -15041.165} C_VEL
LIN {X 0,Y 327.747,Z 499.08,A -85,B 0,C 180,E1 -15043.643,E2 -15043.643} C_VEL
LIN {X 0,Y 328.927,Z 492.721,A -85,B 0,C 180,E1 -15045.736,E2 -15045.736} C_VEL
LIN {X 0,Y 330.614,Z 484.525,A -85,B 0,C 180,E1 -15047.952,E2 -15047.952} C_VEL
LIN {X 0,Y 332.602,Z 474.951,A -85,B 0,C 180,E1 -15050.082,E2 -15050.082} C_VEL
LIN {X 0,Y 334.522,Z 465.157,A -85,B 0,C 180,E1 -15051.895,E2 -15051.895} C_VEL
LIN {X 0,Y 336.705,Z 453.498,A -85,B 0,C 180,E1 -15053.69,E2 -15053.69} C_VEL
LIN {X 0,Y 338.838,Z 441.877,A -85,B 0,C 180,E1 -15055.163,E2 -15055.163} C_VEL
LIN {X 0,Y 340.79,Z 429.346,A -85,B 0,C 180,E1 -15056.484,E2 -15056.484} C_VEL
LIN {X 0,Y 342.666,Z 415.351,A -85,B 0,C 180,E1 -15057.674,E2 -15057.674} C_VEL
LIN {X 0,Y 342.652,Z 412.922,A -85,B 0,C 180,E1 -15057.881,E2 -15057.881} C_VEL
LIN {X 0,Y 339.095,Z 399.372,A -85,B 0,C 180,E1 -15059.229,E2 -15059.229} C_VEL
LIN {X 0,Y 334.303,Z 385.321,A -85,B 0,C 180,E1 -15060.519,E2 -15060.519} C_VEL
LIN {X 0,Y 328.024,Z 370.587,A -85,B 0,C 180,E1 -15061.782,E2 -15061.782} C_VEL
LIN {X 0,Y 326.177,Z 366.4,A -85,B 0,C 180,E1 -15062.114,E2 -15062.114} C_VEL
LIN {X 0,Y 326.095,Z 365.773,A -85,B 0,C 180,E1 -15062.16,E2 -15062.16} C_VEL
LIN {X 0,Y 326.208,Z 363.279,A -85,B 0,C 180,E1 -15065.57,E2 -15065.57} C_VEL
LIN {X 0,Y 326.345,Z 360.831,A -85,B 0,C 180,E1 -15069.17,E2 -15069.17} C_VEL
LIN {X 0,Y 326.457,Z 360.441,A -85,B 0,C 180,E1 -15071.107,E2 -15071.107} C_VEL
LIN {X 0,Y 326.523,Z 360.437,A -85,B 0,C 180,E1 -15074.742,E2 -15074.742} C_VEL
LIN {X 0,Y 326.57,Z 360.432,A -85,B 0,C 180,E1 -15078.375,E2 -15078.375} C_VEL
LIN {X 0,Y 326.622,Z 360.424,A -85,B 0,C 180,E1 -15081.391,E2 -15081.391} C_VEL
LIN {X 0,Y 326.591,Z 360.425,A -85,B 0,C 180,E1 -15083.729,E2 -15083.729} C_VEL
LIN {X 0,Y 325.921,Z 360.513,A -85,B 0,C 180,E1 -15084.758,E2 -15084.758} C_VEL
LIN {X 0,Y 323.066,Z 360.865,A -85,B 0,C 180,E1 -15086.432,E2 -15086.432} C_VEL
LIN {X 0,Y 320.66,Z 361.165,A -85,B 0,C 180,E1 -15087.789,E2 -15087.789} C_VEL
LIN {X 0,Y 319.645,Z 361.293,A -85,B 0,C 180,E1 -15088.839,E2 -15088.839} C_VEL
LIN {X 0,Y 319.571,Z 361.302,A -85,B 0,C 180,E1 -15089.194,E2 -15089.194} C_VEL
LIN {X 0,Y 319.607,Z 361.28,A -85,B 0,C 180,E1 -15092.498,E2 -15092.498} C_VEL
LIN {X 0,Y 319.603,Z 361.296,A -85,B 0,C 180,E1 -15095.304,E2 -15095.304} C_VEL
LIN {X 0,Y 319.594,Z 361.289,A -85,B 0,C 180,E1 -15098.047,E2 -15098.047} C_VEL
LIN {X 0,Y 319.687,Z 361.275,A -85,B 0,C 180,E1 -15100.962,E2 -15100.962} C_VEL
LIN {X 0,Y 319.729,Z 361.271,A -85,B 0,C 180,E1 -15105.275,E2 -15105.275} C_VEL
LIN {X 0,Y 319.758,Z 361.279,A -85,B 0,C 180,E1 -15109.873,E2 -15109.873} C_VEL
LIN {X 0,Y 319.931,Z 361.258,A -85,B 0,C 180,E1 -15112.426,E2 -15112.426} C_VEL
LIN {X 0,Y 319.747,Z 361.281,A -85,B 0,C 180,E1 -15114.956,E2 -15114.956} C_VEL
LIN {X 0,Y 319.99,Z 361.252,A -85,B 0,C 180,E1 -15117.482,E2 -15117.482} C_VEL
LIN {X 0,Y 320.166,Z 361.232,A -85,B 0,C 180,E1 -15120,E2 -15120} C_VEL
LIN {X 0,Y 319.99,Z 361.25,A -85,B 0,C 180,E1 -15122.517,E2 -15122.517} C_VEL
LIN {X 0,Y 319.95,Z 361.257,A -85,B 0,C 180,E1 -15126.305,E2 -15126.305} C_VEL
LIN {X 0,Y 319.84,Z 361.27,A -85,B 0,C 180,E1 -15128.848,E2 -15128.848} C_VEL
LIN {X 0,Y 319.679,Z 361.285,A -85,B 0,C 180,E1 -15132.7,E2 -15132.7} C_VEL
LIN {X 0,Y 319.697,Z 361.284,A -85,B 0,C 180,E1 -15135.296,E2 -15135.296} C_VEL
LIN {X 0,Y 319.672,Z 361.291,A -85,B 0,C 180,E1 -15139.255,E2 -15139.255} C_VEL
LIN {X 0,Y 319.568,Z 361.306,A -85,B 0,C 180,E1 -15143.319,E2 -15143.319} C_VEL
LIN {X 0,Y 319.632,Z 361.3,A -85,B 0,C 180,E1 -15146.088,E2 -15146.088} C_VEL
LIN {X 0,Y 319.587,Z 361.304,A -85,B 0,C 180,E1 -15148.934,E2 -15148.934} C_VEL
LIN {X 0,Y 319.584,Z 361.375,A -85,B 0,C 180,E1 -15152.601,E2 -15152.601} C_VEL
LIN {X 0,Y 320.202,Z 364.915,A -85,B 0,C 180,E1 -15156.342,E2 -15156.342} C_VEL
LIN {X 0,Y 320.818,Z 368.656,A -85,B 0,C 180,E1 -15159.94,E2 -15159.94} C_VEL
LIN {X 0,Y 321.541,Z 373.104,A -85,B 0,C 180,E1 -15163.84,E2 -15163.84} C_VEL
LIN {X 0,Y 321.918,Z 375.809,A -85,B 0,C 180,E1 -15166.091,E2 -15166.091} C_VEL
LIN {X 0,Y 322.009,Z 378.116,A -85,B 0,C 180,E1 -15167.908,E2 -15167.908} C_VEL
LIN {X 0,Y 321.573,Z 381.832,A -85,B 0,C 180,E1 -15170.67,E2 -15170.67} C_VEL
LIN {X 0,Y 320.915,Z 386.636,A -85,B 0,C 180,E1 -15174.125,E2 -15174.125} C_VEL
LIN {X 0,Y 320.297,Z 391.014,A -85,B 0,C 180,E1 -15177.203,E2 -15177.203} C_VEL
LIN {X 0,Y 321.375,Z 394.655,A -85,B 0,C 180,E1 -15177.437,E2 -15177.437} C_VEL
LIN {X 0,Y 326.114,Z 409.225,A -85,B 0,C 180,E1 -15178.485,E2 -15178.485} C_VEL
LIN {X 0,Y 329.847,Z 423.823,A -85,B 0,C 180,E1 -15179.645,E2 -15179.645} C_VEL
LIN {X 0,Y 332.615,Z 439.227,A -85,B 0,C 180,E1 -15181.005,E2 -15181.005} C_VEL
LIN {X 0,Y 333.904,Z 450.604,A -85,B 0,C 180,E1 -15182.13,E2 -15182.13} C_VEL
LIN {X 0,Y 332.73,Z 459.997,A -85,B 0,C 180,E1 -15182.993,E2 -15182.993} C_VEL
LIN {X 0,Y 330.17,Z 473.743,A -85,B 0,C 180,E1 -15184.467,E2 -15184.467} C_VEL
LIN {X 0,Y 327.765,Z 486.219,A -85,B 0,C 180,E1 -15186.127,E2 -15186.127} C_VEL
LIN {X 0,Y 325.692,Z 496.691,A -85,B 0,C 180,E1 -15187.814,E2 -15187.814} C_VEL
LIN {X 0,Y 323.832,Z 506.428,A -85,B 0,C 180,E1 -15189.682,E2 -15189.682} C_VEL
LIN {X 0,Y 321.815,Z 515.992,A -85,B 0,C 180,E1 -15191.869,E2 -15191.869} C_VEL
LIN {X 0,Y 320.382,Z 523.98,A -85,B 0,C 180,E1 -15194.086,E2 -15194.086} C_VEL
LIN {X 0,Y 319.165,Z 531.448,A -85,B 0,C 180,E1 -15196.632,E2 -15196.632} C_VEL
LIN {X 0,Y 318.338,Z 537.382,A -85,B 0,C 180,E1 -15199.185,E2 -15199.185} C_VEL
LIN {X 0,Y 318.06,Z 540.92,A -85,B 0,C 180,E1 -15201.103,E2 -15201.103} C_VEL
LIN {X 0,Y 317.879,Z 544.501,A -85,B 0,C 180,E1 -15203.654,E2 -15203.654} C_VEL
LIN {X 0,Y 317.87,Z 546.86,A -85,B 0,C 180,E1 -15206.197,E2 -15206.197} C_VEL
LIN {X 0,Y 317.89,Z 548.046,A -85,B 0,C 180,E1 -15208.734,E2 -15208.734} C_VEL
LIN {X 0,Y 317.947,Z 548.205,A -85,B 0,C 180,E1 -15210.001,E2 -15210.001} C_VEL
LIN {X 0,Y 317.833,Z 547.587,A -85,B 0,C 180,E1 -15212.535,E2 -15212.535} C_VEL
LIN {X 0,Y 317.868,Z 545.81,A -85,B 0,C 180,E1 -15215.074,E2 -15215.074} C_VEL
LIN {X 0,Y 317.963,Z 542.843,A -85,B 0,C 180,E1 -15217.621,E2 -15217.621} C_VEL
LIN {X 0,Y 318.235,Z 538.621,A -85,B 0,C 180,E1 -15220.177,E2 -15220.177} C_VEL
LIN {X 0,Y 318.937,Z 533.045,A -85,B 0,C 180,E1 -15222.731,E2 -15222.731} C_VEL
LIN {X 0,Y 320.03,Z 525.964,A -85,B 0,C 180,E1 -15225.28,E2 -15225.28} C_VEL
LIN {X 0,Y 321.609,Z 517.169,A -85,B 0,C 180,E1 -15227.815,E2 -15227.815} C_VEL
LIN {X 0,Y 323.501,Z 507.845,A -85,B 0,C 180,E1 -15230.009,E2 -15230.009} C_VEL
LIN {X 0,Y 325.34,Z 498.542,A -85,B 0,C 180,E1 -15231.845,E2 -15231.845} C_VEL
LIN {X 0,Y 327.597,Z 487.134,A -85,B 0,C 180,E1 -15233.719,E2 -15233.719} C_VEL
LIN {X 0,Y 329.951,Z 474.833,A -85,B 0,C 180,E1 -15235.383,E2 -15235.383} C_VEL
LIN {X 0,Y 332.477,Z 461.382,A -85,B 0,C 180,E1 -15236.855,E2 -15236.855} C_VEL
LIN {X 0,Y 333.888,Z 450.465,A -85,B 0,C 180,E1 -15237.865,E2 -15237.865} C_VEL
LIN {X 0,Y 332.149,Z 436.67,A -85,B 0,C 180,E1 -15239.213,E2 -15239.213} C_VEL
LIN {X 0,Y 329.488,Z 422.339,A -85,B 0,C 180,E1 -15240.455,E2 -15240.455} C_VEL
LIN {X 0,Y 325.563,Z 407.463,A -85,B 0,C 180,E1 -15241.627,E2 -15241.627} C_VEL
LIN {X 0,Y 321.166,Z 394.294,A -85,B 0,C 180,E1 -15242.572,E2 -15242.572} C_VEL
LIN {X 0,Y 320.281,Z 390.989,A -85,B 0,C 180,E1 -15242.794,E2 -15242.794} C_VEL
LIN {X 0,Y 321.014,Z 386.094,A -85,B 0,C 180,E1 -15246.237,E2 -15246.237} C_VEL
LIN {X 0,Y 321.704,Z 380.667,A -85,B 0,C 180,E1 -15250.127,E2 -15250.127} C_VEL
LIN {X 0,Y 322.012,Z 377.422,A -85,B 0,C 180,E1 -15252.578,E2 -15252.578} C_VEL
LIN {X 0,Y 321.649,Z 373.667,A -85,B 0,C 180,E1 -15255.638,E2 -15255.638} C_VEL
LIN {X 0,Y 321.013,Z 369.823,A -85,B 0,C 180,E1 -15258.944,E2 -15258.944} C_VEL
LIN {X 0,Y 320.435,Z 366.433,A -85,B 0,C 180,E1 -15262.147,E2 -15262.147} C_VEL
LIN {X 0,Y 319.942,Z 363.436,A -85,B 0,C 180,E1 -15265.171,E2 -15265.171} C_VEL
LIN {X 0,Y 319.577,Z 361.302,A -85,B 0,C 180,E1 -15267.585,E2 -15267.585} C_VEL
LIN {X 0,Y 319.613,Z 361.299,A -85,B 0,C 180,E1 -15271.591,E2 -15271.591} C_VEL
LIN {X 0,Y 319.608,Z 361.3,A -85,B 0,C 180,E1 -15275.304,E2 -15275.304} C_VEL
LIN {X 0,Y 319.601,Z 361.301,A -85,B 0,C 180,E1 -15278.048,E2 -15278.048} C_VEL
LIN {X 0,Y 319.693,Z 361.288,A -85,B 0,C 180,E1 -15280.962,E2 -15280.962} C_VEL
LIN {X 0,Y 319.734,Z 361.286,A -85,B 0,C 180,E1 -15285.276,E2 -15285.276} C_VEL
LIN {X 0,Y 319.761,Z 361.283,A -85,B 0,C 180,E1 -15289.873,E2 -15289.873} C_VEL
LIN {X 0,Y 319.937,Z 361.261,A -85,B 0,C 180,E1 -15292.426,E2 -15292.426} C_VEL
LIN {X 0,Y 319.751,Z 361.282,A -85,B 0,C 180,E1 -15294.956,E2 -15294.956} C_VEL
LIN {X 0,Y 319.995,Z 361.249,A -85,B 0,C 180,E1 -15297.483,E2 -15297.483} C_VEL
LIN {X 0,Y 320.152,Z 361.228,A -85,B 0,C 180,E1 -15300,E2 -15300} C_VEL
LIN {X 0,Y 319.995,Z 361.249,A -85,B 0,C 180,E1 -15302.518,E2 -15302.518} C_VEL
LIN {X 0,Y 319.936,Z 361.252,A -85,B 0,C 180,E1 -15306.638,E2 -15306.638} C_VEL
LIN {X 0,Y 319.761,Z 361.276,A -85,B 0,C 180,E1 -15310.127,E2 -15310.127} C_VEL
LIN {X 0,Y 319.734,Z 361.272,A -85,B 0,C 180,E1 -15314.724,E2 -15314.724} C_VEL
LIN {X 0,Y 319.692,Z 361.272,A -85,B 0,C 180,E1 -15319.038,E2 -15319.038} C_VEL
LIN {X 0,Y 319.565,Z 361.302,A -85,B 0,C 180,E1 -15323.32,E2 -15323.32} C_VEL
LIN {X 0,Y 319.637,Z 361.282,A -85,B 0,C 180,E1 -15326.088,E2 -15326.088} C_VEL
LIN {X 0,Y 319.583,Z 361.293,A -85,B 0,C 180,E1 -15328.934,E2 -15328.934} C_VEL
LIN {X 0,Y 319.533,Z 361.301,A -85,B 0,C 180,E1 -15331.862,E2 -15331.862} C_VEL
LIN {X 0,Y 319.583,Z 361.301,A -85,B 0,C 180,E1 -15335.543,E2 -15335.543} C_VEL
LIN {X 0,Y 319.576,Z 361.304,A -85,B 0,C 180,E1 -15338.008,E2 -15338.008} C_VEL
LIN {X 0,Y 319.528,Z 361.31,A -85,B 0,C 180,E1 -15341.597,E2 -15341.597} C_VEL
LIN {X 0,Y 319.488,Z 361.319,A -85,B 0,C 180,E1 -15345.256,E2 -15345.256} C_VEL
LIN {X 0,Y 319.425,Z 361.327,A -85,B 0,C 180,E1 -15348.695,E2 -15348.695} C_VEL
LIN {X 0,Y 319.319,Z 361.478,A -85,B 0,C 180,E1 -15350.384,E2 -15350.384} C_VEL
LIN {X 0,Y 319.179,Z 364.295,A -85,B 0,C 180,E1 -15354.558,E2 -15354.558} C_VEL
LIN {X 0,Y 319.085,Z 366.179,A -85,B 0,C 180,E1 -15357.16,E2 -15357.16} C_VEL
LIN {X 0,Y 320.273,Z 369.409,A -85,B 0,C 180,E1 -15357.421,E2 -15357.421} C_VEL
LIN {X 0,Y 325.857,Z 381.79,A -85,B 0,C 180,E1 -15358.515,E2 -15358.515} C_VEL
LIN {X 0,Y 331.094,Z 395.936,A -85,B 0,C 180,E1 -15359.843,E2 -15359.843} C_VEL
LIN {X 0,Y 334.81,Z 408.685,A -85,B 0,C 180,E1 -15361.131,E2 -15361.131} C_VEL
LIN {X 0,Y 336.313,Z 416.154,A -85,B 0,C 180,E1 -15361.907,E2 -15361.907} C_VEL
LIN {X 0,Y 334.336,Z 430.224,A -85,B 0,C 180,E1 -15363.131,E2 -15363.131} C_VEL
LIN {X 0,Y 332.077,Z 443.95,A -85,B 0,C 180,E1 -15364.623,E2 -15364.623} C_VEL
LIN {X 0,Y 329.913,Z 455.269,A -85,B 0,C 180,E1 -15366.124,E2 -15366.124} C_VEL
LIN {X 0,Y 327.676,Z 466.681,A -85,B 0,C 180,E1 -15367.954,E2 -15367.954} C_VEL
LIN {X 0,Y 325.66,Z 476.28,A -85,B 0,C 180,E1 -15369.8,E2 -15369.8} C_VEL
LIN {X 0,Y 323.644,Z 485.68,A -85,B 0,C 180,E1 -15371.974,E2 -15371.974} C_VEL
LIN {X 0,Y 321.88,Z 494.145,A -85,B 0,C 180,E1 -15374.373,E2 -15374.373} C_VEL
LIN {X 0,Y 320.527,Z 500.785,A -85,B 0,C 180,E1 -15376.689,E2 -15376.689} C_VEL
LIN {X 0,Y 319.46,Z 506.56,A -85,B 0,C 180,E1 -15379.222,E2 -15379.222} C_VEL
LIN {X 0,Y 318.877,Z 509.976,A -85,B 0,C 180,E1 -15381.125,E2 -15381.125} C_VEL
LIN {X 0,Y 318.384,Z 513.432,A -85,B 0,C 180,E1 -15383.663,E2 -15383.663} C_VEL
LIN {X 0,Y 318.078,Z 515.716,A -85,B 0,C 180,E1 -15386.199,E2 -15386.199} C_VEL
LIN {X 0,Y 317.999,Z 516.879,A -85,B 0,C 180,E1 -15388.733,E2 -15388.733} C_VEL
LIN {X 0,Y 317.999,Z 516.893,A -85,B 0,C 180,E1 -15391.266,E2 -15391.266} C_VEL
LIN {X 0,Y 318.076,Z 515.787,A -85,B 0,C 180,E1 -15393.8,E2 -15393.8} C_VEL
LIN {X 0,Y 318.383,Z 513.557,A -85,B 0,C 180,E1 -15396.336,E2 -15396.336} C_VEL
LIN {X 0,Y 318.864,Z 510.152,A -85,B 0,C 180,E1 -15398.875,E2 -15398.875} C_VEL
LIN {X 0,Y 319.632,Z 505.485,A -85,B 0,C 180,E1 -15401.413,E2 -15401.413} C_VEL
LIN {X 0,Y 320.85,Z 499.427,A -85,B 0,C 180,E1 -15403.942,E2 -15403.942} C_VEL
LIN {X 0,Y 322.144,Z 492.457,A -85,B 0,C 180,E1 -15406.277,E2 -15406.277} C_VEL
LIN {X 0,Y 324.142,Z 483.645,A -85,B 0,C 180,E1 -15408.651,E2 -15408.651} C_VEL
LIN {X 0,Y 326.265,Z 473.817,A -85,B 0,C 180,E1 -15410.819,E2 -15410.819} C_VEL
LIN {X 0,Y 328.521,Z 462.706,A -85,B 0,C 180,E1 -15412.837,E2 -15412.837} C_VEL
LIN {X 0,Y 330.845,Z 450.616,A -85,B 0,C 180,E1 -15414.637,E2 -15414.637} C_VEL
LIN {X 0,Y 333.099,Z 438.365,A -85,B 0,C 180,E1 -15416.131,E2 -15416.131} C_VEL
LIN {X 0,Y 335.208,Z 424.965,A -85,B 0,C 180,E1 -15417.467,E2 -15417.467} C_VEL
LIN {X 0,Y 336.399,Z 415.692,A -85,B 0,C 180,E1 -15418.235,E2 -15418.235} C_VEL
LIN {X 0,Y 333.262,Z 402.87,A -85,B 0,C 180,E1 -15419.578,E2 -15419.578} C_VEL
LIN {X 0,Y 328.551,Z 388.548,A -85,B 0,C 180,E1 -15420.969,E2 -15420.969} C_VEL
LIN {X 0,Y 322.321,Z 373.566,A -85,B 0,C 180,E1 -15422.33,E2 -15422.33} C_VEL
LIN {X 0,Y 319.282,Z 367.229,A -85,B 0,C 180,E1 -15422.879,E2 -15422.879} C_VEL
LIN {X 0,Y 319.079,Z 366.15,A -85,B 0,C 180,E1 -15422.967,E2 -15422.967} C_VEL
LIN {X 0,Y 319.2,Z 363.656,A -85,B 0,C 180,E1 -15426.474,E2 -15426.474} C_VEL
LIN {X 0,Y 319.315,Z 361.534,A -85,B 0,C 180,E1 -15429.663,E2 -15429.663} C_VEL
LIN {X 0,Y 319.477,Z 361.312,A -85,B 0,C 180,E1 -15432.995,E2 -15432.995} C_VEL
LIN {X 0,Y 319.552,Z 361.306,A -85,B 0,C 180,E1 -15437.016,E2 -15437.016} C_VEL
LIN {X 0,Y 319.546,Z 361.308,A -85,B 0,C 180,E1 -15440.371,E2 -15440.371} C_VEL
LIN {X 0,Y 319.556,Z 361.304,A -85,B 0,C 180,E1 -15443.728,E2 -15443.728} C_VEL
LIN {X 0,Y 319.576,Z 361.287,A -85,B 0,C 180,E1 -15446.686,E2 -15446.686} C_VEL
LIN {X 0,Y 319.571,Z 361.302,A -85,B 0,C 180,E1 -15449.194,E2 -15449.194} C_VEL
LIN {X 0,Y 318.946,Z 361.382,A -85,B 0,C 180,E1 -15450.246,E2 -15450.246} C_VEL
LIN {X 0,Y 316.166,Z 361.728,A -85,B 0,C 180,E1 -15451.958,E2 -15451.958} C_VEL
LIN {X 0,Y 313.762,Z 362.024,A -85,B 0,C 180,E1 -15453.345,E2 -15453.345} C_VEL
LIN {X 0,Y 312.687,Z 362.155,A -85,B 0,C 180,E1 -15454.418,E2 -15454.418} C_VEL
LIN {X 0,Y 312.577,Z 362.167,A -85,B 0,C 180,E1 -15454.782,E2 -15454.782} C_VEL
LIN {X 0,Y 312.585,Z 362.166,A -85,B 0,C 180,E1 -15457.529,E2 -15457.529} C_VEL
LIN {X 0,Y 312.636,Z 362.16,A -85,B 0,C 180,E1 -15461.656,E2 -15461.656} C_VEL
LIN {X 0,Y 312.692,Z 362.142,A -85,B 0,C 180,E1 -15465.686,E2 -15465.686} C_VEL
LIN {X 0,Y 312.702,Z 362.156,A -85,B 0,C 180,E1 -15469.642,E2 -15469.642} C_VEL
LIN {X 0,Y 312.87,Z 362.137,A -85,B 0,C 180,E1 -15472.254,E2 -15472.254} C_VEL
LIN {X 0,Y 312.717,Z 362.157,A -85,B 0,C 180,E1 -15474.842,E2 -15474.842} C_VEL
LIN {X 0,Y 312.989,Z 362.124,A -85,B 0,C 180,E1 -15478.713,E2 -15478.713} C_VEL
LIN {X 0,Y 313.118,Z 362.11,A -85,B 0,C 180,E1 -15480,E2 -15480} C_VEL
LIN {X 0,Y 312.936,Z 362.129,A -85,B 0,C 180,E1 -15482.574,E2 -15482.574} C_VEL
LIN {X 0,Y 312.908,Z 362.134,A -85,B 0,C 180,E1 -15486.448,E2 -15486.448} C_VEL
LIN {X 0,Y 312.785,Z 362.149,A -85,B 0,C 180,E1 -15489.049,E2 -15489.049} C_VEL
LIN {X 0,Y 312.632,Z 362.164,A -85,B 0,C 180,E1 -15492.991,E2 -15492.991} C_VEL
LIN {X 0,Y 312.636,Z 362.162,A -85,B 0,C 180,E1 -15495.65,E2 -15495.65} C_VEL
LIN {X 0,Y 312.628,Z 362.168,A -85,B 0,C 180,E1 -15499.237,E2 -15499.237} C_VEL
LIN {X 0,Y 312.543,Z 362.181,A -85,B 0,C 180,E1 -15502.789,E2 -15502.789} C_VEL
LIN {X 0,Y 312.6,Z 362.176,A -85,B 0,C 180,E1 -15505.936,E2 -15505.936} C_VEL
LIN {X 0,Y 312.543,Z 362.181,A -85,B 0,C 180,E1 -15509.65,E2 -15509.65} C_VEL
LIN {X 0,Y 312.505,Z 362.236,A -85,B 0,C 180,E1 -15511.914,E2 -15511.914} C_VEL
LIN {X 0,Y 313.217,Z 366.091,A -85,B 0,C 180,E1 -15516.122,E2 -15516.122} C_VEL
LIN {X 0,Y 313.942,Z 370.537,A -85,B 0,C 180,E1 -15520.481,E2 -15520.481} C_VEL
LIN {X 0,Y 314.667,Z 374.925,A -85,B 0,C 180,E1 -15524.381,E2 -15524.381} C_VEL
LIN {X 0,Y 315.001,Z 378.588,A -85,B 0,C 180,E1 -15527.414,E2 -15527.414} C_VEL
LIN {X 0,Y 314.569,Z 382.545,A -85,B 0,C 180,E1 -15530.452,E2 -15530.452} C_VEL
LIN {X 0,Y 313.934,Z 386.928,A -85,B 0,C 180,E1 -15533.7,E2 -15533.7} C_VEL
LIN {X 0,Y 313.432,Z 390.73,A -85,B 0,C 180,E1 -15536.403,E2 -15536.403} C_VEL
LIN {X 0,Y 314.436,Z 394.146,A -85,B 0,C 180,E1 -15536.622,E2 -15536.622} C_VEL
LIN {X 0,Y 319.367,Z 408.989,A -85,B 0,C 180,E1 -15537.747,E2 -15537.747} C_VEL
LIN {X 0,Y 323.259,Z 424.243,A -85,B 0,C 180,E1 -15539.01,E2 -15539.01} C_VEL
LIN {X 0,Y 325.907,Z 438.977,A -85,B 0,C 180,E1 -15540.359,E2 -15540.359} C_VEL
LIN {X 0,Y 327.367,Z 451.707,A -85,B 0,C 180,E1 -15541.666,E2 -15541.666} C_VEL
LIN {X 0,Y 326.947,Z 455.773,A -85,B 0,C 180,E1 -15542.051,E2 -15542.051} C_VEL
LIN {X 0,Y 324.753,Z 468.206,A -85,B 0,C 180,E1 -15543.318,E2 -15543.318} C_VEL
LIN {X 0,Y 322.351,Z 480.486,A -85,B 0,C 180,E1 -15544.841,E2 -15544.841} C_VEL
LIN {X 0,Y 319.769,Z 492.743,A -85,B 0,C 180,E1 -15546.697,E2 -15546.697} C_VEL
LIN {X 0,Y 317.551,Z 503.647,A -85,B 0,C 180,E1 -15548.713,E2 -15548.713} C_VEL
LIN {X 0,Y 315.521,Z 513.127,A -85,B 0,C 180,E1 -15550.82,E2 -15550.82} C_VEL
LIN {X 0,Y 313.865,Z 521.513,A -85,B 0,C 180,E1 -15553.077,E2 -15553.077} C_VEL
LIN {X 0,Y 312.428,Z 529.403,A -85,B 0,C 180,E1 -15555.674,E2 -15555.674} C_VEL
LIN {X 0,Y 311.523,Z 535.695,A -85,B 0,C 180,E1 -15558.286,E2 -15558.286} C_VEL
LIN {X 0,Y 310.982,Z 540.57,A -85,B 0,C 180,E1 -15560.898,E2 -15560.898} C_VEL
LIN {X 0,Y 310.804,Z 544.152,A -85,B 0,C 180,E1 -15563.509,E2 -15563.509} C_VEL
LIN {X 0,Y 310.776,Z 546.512,A -85,B 0,C 180,E1 -15566.11,E2 -15566.11} C_VEL
LIN {X 0,Y 310.795,Z 547.699,A -85,B 0,C 180,E1 -15568.705,E2 -15568.705} C_VEL
LIN {X 0,Y 310.854,Z 547.857,A -85,B 0,C 180,E1 -15570.001,E2 -15570.001} C_VEL
LIN {X 0,Y 310.753,Z 547.24,A -85,B 0,C 180,E1 -15572.593,E2 -15572.593} C_VEL
LIN {X 0,Y 310.789,Z 545.462,A -85,B 0,C 180,E1 -15575.19,E2 -15575.19} C_VEL
LIN {X 0,Y 310.882,Z 542.492,A -85,B 0,C 180,E1 -15577.796,E2 -15577.796} C_VEL
LIN {X 0,Y 311.167,Z 538.268,A -85,B 0,C 180,E1 -15580.41,E2 -15580.41} C_VEL
LIN {X 0,Y 311.926,Z 532.692,A -85,B 0,C 180,E1 -15583.022,E2 -15583.022} C_VEL
LIN {X 0,Y 313.123,Z 525.611,A -85,B 0,C 180,E1 -15585.625,E2 -15585.625} C_VEL
LIN {X 0,Y 314.763,Z 516.815,A -85,B 0,C 180,E1 -15588.216,E2 -15588.216} C_VEL
LIN {X 0,Y 316.762,Z 507.49,A -85,B 0,C 180,E1 -15590.454,E2 -15590.454} C_VEL
LIN {X 0,Y 318.702,Z 498.017,A -85,B 0,C 180,E1 -15592.359,E2 -15592.359} C_VEL
LIN {X 0,Y 321.186,Z 485.744,A -85,B 0,C 180,E1 -15594.395,E2 -15594.395} C_VEL
LIN {X 0,Y 323.759,Z 473.249,A -85,B 0,C 180,E1 -15596.077,E2 -15596.077} C_VEL
LIN {X 0,Y 326.276,Z 460.139,A -85,B 0,C 180,E1 -15597.512,E2 -15597.512} C_VEL
LIN {X 0,Y 327.349,Z 451.563,A -85,B 0,C 180,E1 -15598.328,E2 -15598.328} C_VEL
LIN {X 0,Y 325.881,Z 439.074,A -85,B 0,C 180,E1 -15599.613,E2 -15599.613} C_VEL
LIN {X 0,Y 323.471,Z 425.301,A -85,B 0,C 180,E1 -15600.873,E2 -15600.873} C_VEL
LIN {X 0,Y 319.897,Z 410.872,A -85,B 0,C 180,E1 -15602.076,E2 -15602.076} C_VEL
LIN {X 0,Y 315.417,Z 397.067,A -85,B 0,C 180,E1 -15603.143,E2 -15603.143} C_VEL
LIN {X 0,Y 313.559,Z 391.708,A -85,B 0,C 180,E1 -15603.528,E2 -15603.528} C_VEL
LIN {X 0,Y 313.421,Z 390.621,A -85,B 0,C 180,E1 -15603.59,E2 -15603.59} C_VEL
LIN {X 0,Y 314.093,Z 385.722,A -85,B 0,C 180,E1 -15607.168,E2 -15607.168} C_VEL
LIN {X 0,Y 314.772,Z 381.07,A -85,B 0,C 180,E1 -15610.613,E2 -15610.613} C_VEL
LIN {X 0,Y 315.001,Z 378.52,A -85,B 0,C 180,E1 -15612.586,E2 -15612.586} C_VEL
LIN {X 0,Y 314.666,Z 374.876,A -85,B 0,C 180,E1 -15615.62,E2 -15615.62} C_VEL
LIN {X 0,Y 313.937,Z 370.454,A -85,B 0,C 180,E1 -15619.566,E2 -15619.566} C_VEL
LIN {X 0,Y 313.36,Z 367.237,A -85,B 0,C 180,E1 -15622.732,E2 -15622.732} C_VEL
LIN {X 0,Y 312.785,Z 363.827,A -85,B 0,C 180,E1 -15626.239,E2 -15626.239} C_VEL
LIN {X 0,Y 312.502,Z 362.186,A -85,B 0,C 180,E1 -15628.273,E2 -15628.273} C_VEL
LIN {X 0,Y 312.572,Z 362.176,A -85,B 0,C 180,E1 -15631.825,E2 -15631.825} C_VEL
LIN {X 0,Y 312.588,Z 362.175,A -85,B 0,C 180,E1 -15634.711,E2 -15634.711} C_VEL
LIN {X 0,Y 312.59,Z 362.174,A -85,B 0,C 180,E1 -15637.529,E2 -15637.529} C_VEL
LIN {X 0,Y 312.642,Z 362.168,A -85,B 0,C 180,E1 -15641.657,E2 -15641.657} C_VEL
LIN {X 0,Y 312.697,Z 362.164,A -85,B 0,C 180,E1 -15645.686,E2 -15645.686} C_VEL
LIN {X 0,Y 312.705,Z 362.162,A -85,B 0,C 180,E1 -15649.642,E2 -15649.642} C_VEL
LIN {X 0,Y 312.875,Z 362.142,A -85,B 0,C 180,E1 -15652.254,E2 -15652.254} C_VEL
LIN {X 0,Y 312.721,Z 362.157,A -85,B 0,C 180,E1 -15654.843,E2 -15654.843} C_VEL
LIN {X 0,Y 312.992,Z 362.122,A -85,B 0,C 180,E1 -15658.714,E2 -15658.714} C_VEL
LIN {X 0,Y 312.994,Z 362.124,A -85,B 0,C 180,E1 -15661.287,E2 -15661.287} C_VEL
LIN {X 0,Y 312.721,Z 362.156,A -85,B 0,C 180,E1 -15665.158,E2 -15665.158} C_VEL
LIN {X 0,Y 312.876,Z 362.136,A -85,B 0,C 180,E1 -15667.746,E2 -15667.746} C_VEL
LIN {X 0,Y 312.673,Z 362.139,A -85,B 0,C 180,E1 -15671.671,E2 -15671.671} C_VEL
LIN {X 0,Y 312.703,Z 362.148,A -85,B 0,C 180,E1 -15674.888,E2 -15674.888} C_VEL
LIN {X 0,Y 312.612,Z 362.15,A -85,B 0,C 180,E1 -15679.225,E2 -15679.225} C_VEL
LIN {X 0,Y 312.531,Z 362.174,A -85,B 0,C 180,E1 -15682.781,E2 -15682.781} C_VEL
LIN {X 0,Y 312.605,Z 362.158,A -85,B 0,C 180,E1 -15685.935,E2 -15685.935} C_VEL
LIN {X 0,Y 312.541,Z 362.177,A -85,B 0,C 180,E1 -15689.651,E2 -15689.651} C_VEL
LIN {X 0,Y 312.522,Z 362.164,A -85,B 0,C 180,E1 -15693.689,E2 -15693.689} C_VEL
LIN {X 0,Y 312.54,Z 362.18,A -85,B 0,C 180,E1 -15697.383,E2 -15697.383} C_VEL
LIN {X 0,Y 312.493,Z 362.188,A -85,B 0,C 180,E1 -15700.709,E2 -15700.709} C_VEL
LIN {X 0,Y 312.453,Z 362.194,A -85,B 0,C 180,E1 -15704.21,E2 -15704.21} C_VEL
LIN {X 0,Y 312.399,Z 362.202,A -85,B 0,C 180,E1 -15707.936,E2 -15707.936} C_VEL
LIN {X 0,Y 312.272,Z 362.238,A -85,B 0,C 180,E1 -15709.925,E2 -15709.925} C_VEL
LIN {X 0,Y 312.192,Z 363.95,A -85,B 0,C 180,E1 -15712.567,E2 -15712.567} C_VEL
LIN {X 0,Y 312.063,Z 366.547,A -85,B 0,C 180,E1 -15716.305,E2 -15716.305} C_VEL
LIN {X 0,Y 313.268,Z 369.883,A -85,B 0,C 180,E1 -15716.599,E2 -15716.599} C_VEL
LIN {X 0,Y 314.521,Z 372.32,A -85,B 0,C 180,E1 -15716.83,E2 -15716.83} C_VEL
LIN {X 0,Y 320.346,Z 385.548,A -85,B 0,C 180,E1 -15718.085,E2 -15718.085} C_VEL
LIN {X 0,Y 324.852,Z 398.044,A -85,B 0,C 180,E1 -15719.32,E2 -15719.32} C_VEL
LIN {X 0,Y 328.518,Z 410.82,A -85,B 0,C 180,E1 -15720.665,E2 -15720.665} C_VEL
LIN {X 0,Y 329.822,Z 416.522,A -85,B 0,C 180,E1 -15721.303,E2 -15721.303} C_VEL
LIN {X 0,Y 329.212,Z 423.094,A -85,B 0,C 180,E1 -15721.88,E2 -15721.88} C_VEL
LIN {X 0,Y 327.037,Z 436.389,A -85,B 0,C 180,E1 -15723.173,E2 -15723.173} C_VEL
LIN {X 0,Y 324.746,Z 449.043,A -85,B 0,C 180,E1 -15724.695,E2 -15724.695} C_VEL
LIN {X 0,Y 322.523,Z 460.07,A -85,B 0,C 180,E1 -15726.299,E2 -15726.299} C_VEL
LIN {X 0,Y 320.335,Z 470.42,A -85,B 0,C 180,E1 -15728.1,E2 -15728.1} C_VEL
LIN {X 0,Y 318.323,Z 479.544,A -85,B 0,C 180,E1 -15729.988,E2 -15729.988} C_VEL
LIN {X 0,Y 316.338,Z 488.457,A -85,B 0,C 180,E1 -15732.212,E2 -15732.212} C_VEL
LIN {X 0,Y 314.776,Z 495.832,A -85,B 0,C 180,E1 -15734.459,E2 -15734.459} C_VEL
LIN {X 0,Y 313.234,Z 502.726,A -85,B 0,C 180,E1 -15737.034,E2 -15737.034} C_VEL
LIN {X 0,Y 312.259,Z 508.129,A -85,B 0,C 180,E1 -15739.626,E2 -15739.626} C_VEL
LIN {X 0,Y 311.526,Z 512.206,A -85,B 0,C 180,E1 -15742.22,E2 -15742.22} C_VEL
LIN {X 0,Y 311.165,Z 515.064,A -85,B 0,C 180,E1 -15744.816,E2 -15744.816} C_VEL
LIN {X 0,Y 310.941,Z 516.783,A -85,B 0,C 180,E1 -15747.409,E2 -15747.409} C_VEL
LIN {X 0,Y 310.9,Z 517.381,A -85,B 0,C 180,E1 -15749.999,E2 -15749.999} C_VEL
LIN {X 0,Y 310.94,Z 516.825,A -85,B 0,C 180,E1 -15752.59,E2 -15752.59} C_VEL
LIN {X 0,Y 311.164,Z 515.161,A -85,B 0,C 180,E1 -15755.183,E2 -15755.183} C_VEL
LIN {X 0,Y 311.523,Z 512.355,A -85,B 0,C 180,E1 -15757.779,E2 -15757.779} C_VEL
LIN {X 0,Y 312.214,Z 508.33,A -85,B 0,C 180,E1 -15760.374,E2 -15760.374} C_VEL
LIN {X 0,Y 313.191,Z 502.99,A -85,B 0,C 180,E1 -15762.967,E2 -15762.967} C_VEL
LIN {X 0,Y 314.743,Z 496.168,A -85,B 0,C 180,E1 -15765.542,E2 -15765.542} C_VEL
LIN {X 0,Y 316.243,Z 488.838,A -85,B 0,C 180,E1 -15767.792,E2 -15767.792} C_VEL
LIN {X 0,Y 318.279,Z 479.983,A -85,B 0,C 180,E1 -15770.014,E2 -15770.014} C_VEL
LIN {X 0,Y 320.221,Z 470.952,A -85,B 0,C 180,E1 -15771.907,E2 -15771.907} C_VEL
LIN {X 0,Y 322.489,Z 460.428,A -85,B 0,C 180,E1 -15773.75,E2 -15773.75} C_VEL
LIN {X 0,Y 324.838,Z 448.63,A -85,B 0,C 180,E1 -15775.467,E2 -15775.467} C_VEL
LIN {X 0,Y 327.133,Z 435.893,A -85,B 0,C 180,E1 -15776.99,E2 -15776.99} C_VEL
LIN {X 0,Y 329.308,Z 422.804,A -85,B 0,C 180,E1 -15778.252,E2 -15778.252} C_VEL
LIN {X 0,Y 329.996,Z 417.503,A -85,B 0,C 180,E1 -15778.705,E2 -15778.705} C_VEL
LIN {X 0,Y 327.285,Z 406.008,A -85,B 0,C 180,E1 -15779.957,E2 -15779.957} C_VEL
LIN {X 0,Y 323.166,Z 393.069,A -85,B 0,C 180,E1 -15781.292,E2 -15781.292} C_VEL
LIN {X 0,Y 318.125,Z 380.193,A -85,B 0,C 180,E1 -15782.547,E2 -15782.547} C_VEL
LIN {X 0,Y 313.255,Z 369.849,A -85,B 0,C 180,E1 -15783.521,E2 -15783.521} C_VEL
LIN {X 0,Y 312.19,Z 367.292,A -85,B 0,C 180,E1 -15783.736,E2 -15783.736} C_VEL
LIN {X 0,Y 312.057,Z 366.529,A -85,B 0,C 180,E1 -15783.82,E2 -15783.82} C_VEL
LIN {X 0,Y 312.207,Z 364.036,A -85,B 0,C 180,E1 -15787.429,E2 -15787.429} C_VEL
LIN {X 0,Y 312.268,Z 362.324,A -85,B 0,C 180,E1 -15790.074,E2 -15790.074} C_VEL
LIN {X 0,Y 312.404,Z 362.191,A -85,B 0,C 180,E1 -15792.445,E2 -15792.445} C_VEL
LIN {X 0,Y 312.456,Z 362.191,A -85,B 0,C 180,E1 -15796.034,E2 -15796.034} C_VEL
LIN {X 0,Y 312.502,Z 362.184,A -85,B 0,C 180,E1 -15799.874,E2 -15799.874} C_VEL
LIN {X 0,Y 312.536,Z 362.179,A -85,B 0,C 180,E1 -15802.616,E2 -15802.616} C_VEL
LIN {X 0,Y 312.518,Z 362.168,A -85,B 0,C 180,E1 -15806.311,E2 -15806.311} C_VEL
LIN {X 0,Y 312.544,Z 362.177,A -85,B 0,C 180,E1 -15810.35,E2 -15810.35} C_VEL
LIN {X 0,Y 312.601,Z 362.158,A -85,B 0,C 180,E1 -15814.064,E2 -15814.064} C_VEL
LIN {X 0,Y 312.577,Z 362.167,A -85,B 0,C 180,E1 -15814.782,E2 -15814.782} C_VEL
LIN {X 0,Y 311.837,Z 362.267,A -85,B 0,C 180,E1 -15815.858,E2 -15815.858} C_VEL
LIN {X 0,Y 308.937,Z 362.62,A -85,B 0,C 180,E1 -15817.608,E2 -15817.608} C_VEL
LIN {X 0,Y 306.563,Z 362.903,A -85,B 0,C 180,E1 -15819.028,E2 -15819.028} C_VEL
LIN {X 0,Y 305.612,Z 363.018,A -85,B 0,C 180,E1 -15820.128,E2 -15820.128} C_VEL
LIN {X 0,Y 305.568,Z 363.026,A -85,B 0,C 180,E1 -15820.5,E2 -15820.5} C_VEL
LIN {X 0,Y 305.592,Z 363.042,A -85,B 0,C 180,E1 -15823.98,E2 -15823.98} C_VEL
LIN {X 0,Y 305.588,Z 363.017,A -85,B 0,C 180,E1 -15826.704,E2 -15826.704} C_VEL
LIN {X 0,Y 305.794,Z 363.02,A -85,B 0,C 180,E1 -15831.207,E2 -15831.207} C_VEL
LIN {X 0,Y 305.851,Z 363.012,A -85,B 0,C 180,E1 -15833.402,E2 -15833.402} C_VEL
LIN {X 0,Y 305.956,Z 363,A -85,B 0,C 180,E1 -15838.684,E2 -15838.684} C_VEL
LIN {X 0,Y 305.955,Z 363.001,A -85,B 0,C 180,E1 -15841.316,E2 -15841.316} C_VEL
LIN {X 0,Y 305.85,Z 363.013,A -85,B 0,C 180,E1 -15846.597,E2 -15846.597} C_VEL
LIN {X 0,Y 305.733,Z 363.029,A -85,B 0,C 180,E1 -15849.26,E2 -15849.26} C_VEL
LIN {X 0,Y 305.586,Z 363.042,A -85,B 0,C 180,E1 -15853.296,E2 -15853.296} C_VEL
LIN {X 0,Y 305.591,Z 363.041,A -85,B 0,C 180,E1 -15856.02,E2 -15856.02} C_VEL
LIN {X 0,Y 305.574,Z 363.047,A -85,B 0,C 180,E1 -15859.445,E2 -15859.445} C_VEL
LIN {X 0,Y 305.488,Z 363.06,A -85,B 0,C 180,E1 -15863.042,E2 -15863.042} C_VEL
LIN {X 0,Y 305.545,Z 363.054,A -85,B 0,C 180,E1 -15866.227,E2 -15866.227} C_VEL
LIN {X 0,Y 305.493,Z 363.06,A -85,B 0,C 180,E1 -15869.05,E2 -15869.05} C_VEL
LIN {X 0,Y 305.494,Z 363.229,A -85,B 0,C 180,E1 -15871.357,E2 -15871.357} C_VEL
LIN {X 0,Y 306.032,Z 366.462,A -85,B 0,C 180,E1 -15875.038,E2 -15875.038} C_VEL
LIN {X 0,Y 306.684,Z 370.108,A -85,B 0,C 180,E1 -15878.818,E2 -15878.818} C_VEL
LIN {X 0,Y 307.148,Z 372.994,A -85,B 0,C 180,E1 -15881.572,E2 -15881.572} C_VEL
LIN {X 0,Y 307.884,Z 377.898,A -85,B 0,C 180,E1 -15885.915,E2 -15885.915} C_VEL
LIN {X 0,Y 307.854,Z 381.101,A -85,B 0,C 180,E1 -15888.545,E2 -15888.545} C_VEL
LIN {X 0,Y 307.238,Z 385.386,A -85,B 0,C 180,E1 -15891.858,E2 -15891.858} C_VEL
LIN {X 0,Y 306.52,Z 390.232,A -85,B 0,C 180,E1 -15895.515,E2 -15895.515} C_VEL
LIN {X 0,Y 307.418,Z 393.513,A -85,B 0,C 180,E1 -15895.748,E2 -15895.748} C_VEL
LIN {X 0,Y 311.759,Z 405.951,A -85,B 0,C 180,E1 -15896.742,E2 -15896.742} C_VEL
LIN {X 0,Y 315.599,Z 419.916,A -85,B 0,C 180,E1 -15897.928,E2 -15897.928} C_VEL
LIN {X 0,Y 318.266,Z 432.516,A -85,B 0,C 180,E1 -15899.086,E2 -15899.086} C_VEL
LIN {X 0,Y 320.172,Z 445.786,A -85,B 0,C 180,E1 -15900.415,E2 -15900.415} C_VEL
LIN {X 0,Y 320.884,Z 454.18,A -85,B 0,C 180,E1 -15901.335,E2 -15901.335} C_VEL
LIN {X 0,Y 318.669,Z 466.53,A -85,B 0,C 180,E1 -15902.589,E2 -15902.589} C_VEL
LIN {X 0,Y 315.898,Z 480.139,A -85,B 0,C 180,E1 -15904.29,E2 -15904.29} C_VEL
LIN {X 0,Y 313.193,Z 492.393,A -85,B 0,C 180,E1 -15906.177,E2 -15906.177} C_VEL
LIN {X 0,Y 310.817,Z 503.417,A -85,B 0,C 180,E1 -15908.256,E2 -15908.256} C_VEL
LIN {X 0,Y 308.773,Z 512.779,A -85,B 0,C 180,E1 -15910.384,E2 -15910.384} C_VEL
LIN {X 0,Y 306.989,Z 521.162,A -85,B 0,C 180,E1 -15912.686,E2 -15912.686} C_VEL
LIN {X 0,Y 305.656,Z 527.98,A -85,B 0,C 180,E1 -15914.952,E2 -15914.952} C_VEL
LIN {X 0,Y 304.715,Z 533.895,A -85,B 0,C 180,E1 -15917.344,E2 -15917.344} C_VEL
LIN {X 0,Y 304.004,Z 539.129,A -85,B 0,C 180,E1 -15920.016,E2 -15920.016} C_VEL
LIN {X 0,Y 303.799,Z 542.169,A -85,B 0,C 180,E1 -15922.022,E2 -15922.022} C_VEL
LIN {X 0,Y 303.684,Z 545.132,A -85,B 0,C 180,E1 -15924.689,E2 -15924.689} C_VEL
LIN {X 0,Y 303.673,Z 546.901,A -85,B 0,C 180,E1 -15927.348,E2 -15927.348} C_VEL
LIN {X 0,Y 303.762,Z 547.51,A -85,B 0,C 180,E1 -15930.001,E2 -15930.001} C_VEL
LIN {X 0,Y 303.675,Z 546.892,A -85,B 0,C 180,E1 -15932.654,E2 -15932.654} C_VEL
LIN {X 0,Y 303.704,Z 545.112,A -85,B 0,C 180,E1 -15935.312,E2 -15935.312} C_VEL
LIN {X 0,Y 303.802,Z 542.141,A -85,B 0,C 180,E1 -15937.979,E2 -15937.979} C_VEL
LIN {X 0,Y 304.113,Z 537.916,A -85,B 0,C 180,E1 -15940.655,E2 -15940.655} C_VEL
LIN {X 0,Y 304.928,Z 532.338,A -85,B 0,C 180,E1 -15943.326,E2 -15943.326} C_VEL
LIN {X 0,Y 306.223,Z 525.258,A -85,B 0,C 180,E1 -15945.987,E2 -15945.987} C_VEL
LIN {X 0,Y 307.912,Z 516.459,A -85,B 0,C 180,E1 -15948.636,E2 -15948.636} C_VEL
LIN {X 0,Y 310.03,Z 507.135,A -85,B 0,C 180,E1 -15950.919,E2 -15950.919} C_VEL
LIN {X 0,Y 312.054,Z 497.662,A -85,B 0,C 180,E1 -15952.862,E2 -15952.862} C_VEL
LIN {X 0,Y 314.694,Z 485.39,A -85,B 0,C 180,E1 -15954.932,E2 -15954.932} C_VEL
LIN {X 0,Y 317.369,Z 472.896,A -85,B 0,C 180,E1 -15956.643,E2 -15956.643} C_VEL
LIN {X 0,Y 319.844,Z 460.38,A -85,B 0,C 180,E1 -15958.043,E2 -15958.043} C_VEL
LIN {X 0,Y 320.865,Z 454.047,A -85,B 0,C 180,E1 -15958.659,E2 -15958.659} C_VEL
LIN {X 0,Y 319.708,Z 442.268,A -85,B 0,C 180,E1 -15959.924,E2 -15959.924} C_VEL
LIN {X 0,Y 317.642,Z 429.203,A -85,B 0,C 180,E1 -15961.204,E2 -15961.204} C_VEL
LIN {X 0,Y 314.273,Z 414.494,A -85,B 0,C 180,E1 -15962.517,E2 -15962.517} C_VEL
LIN {X 0,Y 309.839,Z 400.189,A -85,B 0,C 180,E1 -15963.704,E2 -15963.704} C_VEL
LIN {X 0,Y 306.621,Z 391.085,A -85,B 0,C 180,E1 -15964.397,E2 -15964.397} C_VEL
LIN {X 0,Y 306.514,Z 390.216,A -85,B 0,C 180,E1 -15964.473,E2 -15964.473} C_VEL
LIN {X 0,Y 307.208,Z 385.346,A -85,B 0,C 180,E1 -15968.148,E2 -15968.148} C_VEL
LIN {X 0,Y 307.85,Z 381.03,A -85,B 0,C 180,E1 -15971.457,E2 -15971.457} C_VEL
LIN {X 0,Y 307.874,Z 377.793,A -85,B 0,C 180,E1 -15974.084,E2 -15974.084} C_VEL
LIN {X 0,Y 307.356,Z 374.49,A -85,B 0,C 180,E1 -15977.031,E2 -15977.031} C_VEL
LIN {X 0,Y 306.859,Z 371.208,A -85,B 0,C 180,E1 -15980.112,E2 -15980.112} C_VEL
LIN {X 0,Y 306.3,Z 367.878,A -85,B 0,C 180,E1 -15983.425,E2 -15983.425} C_VEL
LIN {X 0,Y 305.791,Z 365.011,A -85,B 0,C 180,E1 -15986.524,E2 -15986.524} C_VEL
LIN {X 0,Y 305.495,Z 363.055,A -85,B 0,C 180,E1 -15988.962,E2 -15988.962} C_VEL
LIN {X 0,Y 305.521,Z 363.055,A -85,B 0,C 180,E1 -15992.609,E2 -15992.609} C_VEL
LIN {X 0,Y 305.511,Z 363.057,A -85,B 0,C 180,E1 -15995.539,E2 -15995.539} C_VEL
LIN {X 0,Y 305.524,Z 363.054,A -85,B 0,C 180,E1 -15999.815,E2 -15999.815} C_VEL
LIN {X 0,Y 305.578,Z 363.048,A -85,B 0,C 180,E1 -16002.603,E2 -16002.603} C_VEL
LIN {X 0,Y 305.652,Z 363.041,A -85,B 0,C 180,E1 -16005.349,E2 -16005.349} C_VEL
LIN {X 0,Y 305.642,Z 363.043,A -85,B 0,C 180,E1 -16009.4,E2 -16009.4} C_VEL
LIN {X 0,Y 305.816,Z 363.021,A -85,B 0,C 180,E1 -16012.075,E2 -16012.075} C_VEL
LIN {X 0,Y 305.693,Z 363.033,A -85,B 0,C 180,E1 -16014.724,E2 -16014.724} C_VEL
LIN {X 0,Y 305.959,Z 362.998,A -85,B 0,C 180,E1 -16018.684,E2 -16018.684} C_VEL
LIN {X 0,Y 305.961,Z 363,A -85,B 0,C 180,E1 -16021.316,E2 -16021.316} C_VEL
LIN {X 0,Y 305.856,Z 363.006,A -85,B 0,C 180,E1 -16026.598,E2 -16026.598} C_VEL
LIN {X 0,Y 305.739,Z 363.026,A -85,B 0,C 180,E1 -16029.26,E2 -16029.26} C_VEL
LIN {X 0,Y 305.591,Z 363.014,A -85,B 0,C 180,E1 -16033.296,E2 -16033.296} C_VEL
LIN {X 0,Y 305.597,Z 363.041,A -85,B 0,C 180,E1 -16036.02,E2 -16036.02} C_VEL
LIN {X 0,Y 305.564,Z 363.025,A -85,B 0,C 180,E1 -16039.436,E2 -16039.436} C_VEL
LIN {X 0,Y 305.489,Z 363.054,A -85,B 0,C 180,E1 -16043.039,E2 -16043.039} C_VEL
LIN {X 0,Y 305.534,Z 363.036,A -85,B 0,C 180,E1 -16046.221,E2 -16046.221} C_VEL
LIN {X 0,Y 305.491,Z 363.049,A -85,B 0,C 180,E1 -16049.047,E2 -16049.047} C_VEL
LIN {X 0,Y 305.445,Z 363.055,A -85,B 0,C 180,E1 -16051.952,E2 -16051.952} C_VEL
LIN {X 0,Y 305.466,Z 363.055,A -85,B 0,C 180,E1 -16055.113,E2 -16055.113} C_VEL
LIN {X 0,Y 305.47,Z 363.06,A -85,B 0,C 180,E1 -16058.533,E2 -16058.533} C_VEL
LIN {X 0,Y 305.458,Z 363.064,A -85,B 0,C 180,E1 -16062.586,E2 -16062.586} C_VEL
LIN {X 0,Y 305.382,Z 363.076,A -85,B 0,C 180,E1 -16066.336,E2 -16066.336} C_VEL
LIN {X 0,Y 305.274,Z 363.088,A -85,B 0,C 180,E1 -16069.44,E2 -16069.44} C_VEL
LIN {X 0,Y 305.132,Z 365.433,A -85,B 0,C 180,E1 -16073.212,E2 -16073.212} C_VEL
LIN {X 0,Y 305.07,Z 366.969,A -85,B 0,C 180,E1 -16075.452,E2 -16075.452} C_VEL
LIN {X 0,Y 306.209,Z 370.104,A -85,B 0,C 180,E1 -16075.717,E2 -16075.717} C_VEL
LIN {X 0,Y 310.797,Z 379.519,A -85,B 0,C 180,E1 -16076.658,E2 -16076.658} C_VEL
LIN {X 0,Y 316.414,Z 393.482,A -85,B 0,C 180,E1 -16078.08,E2 -16078.08} C_VEL
LIN {X 0,Y 320.456,Z 406.23,A -85,B 0,C 180,E1 -16079.439,E2 -16079.439} C_VEL
LIN {X 0,Y 323.517,Z 418.781,A -85,B 0,C 180,E1 -16080.867,E2 -16080.867} C_VEL
LIN {X 0,Y 321.501,Z 432.481,A -85,B 0,C 180,E1 -16082.143,E2 -16082.143} C_VEL
LIN {X 0,Y 319.085,Z 445.898,A -85,B 0,C 180,E1 -16083.687,E2 -16083.687} C_VEL
LIN {X 0,Y 316.537,Z 458.134,A -85,B 0,C 180,E1 -16085.41,E2 -16085.41} C_VEL
LIN {X 0,Y 314.166,Z 469.144,A -85,B 0,C 180,E1 -16087.301,E2 -16087.301} C_VEL
LIN {X 0,Y 311.649,Z 479.895,A -85,B 0,C 180,E1 -16089.54,E2 -16089.54} C_VEL
LIN {X 0,Y 309.557,Z 488.809,A -85,B 0,C 180,E1 -16091.809,E2 -16091.809} C_VEL
LIN {X 0,Y 307.918,Z 496.183,A -85,B 0,C 180,E1 -16094.104,E2 -16094.104} C_VEL
LIN {X 0,Y 306.298,Z 503.077,A -85,B 0,C 180,E1 -16096.735,E2 -16096.735} C_VEL
LIN {X 0,Y 305.257,Z 508.479,A -85,B 0,C 180,E1 -16099.386,E2 -16099.386} C_VEL
LIN {X 0,Y 304.483,Z 512.556,A -85,B 0,C 180,E1 -16102.039,E2 -16102.039} C_VEL
LIN {X 0,Y 304.094,Z 515.412,A -85,B 0,C 180,E1 -16104.695,E2 -16104.695} C_VEL
LIN {X 0,Y 303.857,Z 517.131,A -85,B 0,C 180,E1 -16107.348,E2 -16107.348} C_VEL
LIN {X 0,Y 303.81,Z 517.729,A -85,B 0,C 180,E1 -16109.999,E2 -16109.999} C_VEL
LIN {X 0,Y 303.856,Z 517.172,A -85,B 0,C 180,E1 -16112.651,E2 -16112.651} C_VEL
LIN {X 0,Y 304.095,Z 515.508,A -85,B 0,C 180,E1 -16115.304,E2 -16115.304} C_VEL
LIN {X 0,Y 304.48,Z 512.703,A -85,B 0,C 180,E1 -16117.96,E2 -16117.96} C_VEL
LIN {X 0,Y 305.219,Z 508.678,A -85,B 0,C 180,E1 -16120.614,E2 -16120.614} C_VEL
LIN {X 0,Y 306.252,Z 503.338,A -85,B 0,C 180,E1 -16123.266,E2 -16123.266} C_VEL
LIN {X 0,Y 307.882,Z 496.515,A -85,B 0,C 180,E1 -16125.897,E2 -16125.897} C_VEL
LIN {X 0,Y 309.468,Z 489.185,A -85,B 0,C 180,E1 -16128.195,E2 -16128.195} C_VEL
LIN {X 0,Y 311.607,Z 480.33,A -85,B 0,C 180,E1 -16130.461,E2 -16130.461} C_VEL
LIN {X 0,Y 314.055,Z 469.684,A -85,B 0,C 180,E1 -16132.707,E2 -16132.707} C_VEL
LIN {X 0,Y 316.489,Z 458.384,A -85,B 0,C 180,E1 -16134.661,E2 -16134.661} C_VEL
LIN {X 0,Y 318.992,Z 446.64,A -85,B 0,C 180,E1 -16136.32,E2 -16136.32} C_VEL
LIN {X 0,Y 321.098,Z 434.819,A -85,B 0,C 180,E1 -16137.716,E2 -16137.716} C_VEL
LIN {X 0,Y 323.255,Z 421.651,A -85,B 0,C 180,E1 -16138.981,E2 -16138.981} C_VEL
LIN {X 0,Y 323.604,Z 419.159,A -85,B 0,C 180,E1 -16139.2,E2 -16139.2} C_VEL
LIN {X 0,Y 320.747,Z 407.055,A -85,B 0,C 180,E1 -16140.576,E2 -16140.576} C_VEL
LIN {X 0,Y 316.298,Z 393.155,A -85,B 0,C 180,E1 -16142.07,E2 -16142.07} C_VEL
LIN {X 0,Y 310.94,Z 379.91,A -85,B 0,C 180,E1 -16143.426,E2 -16143.426} C_VEL
LIN {X 0,Y 306.113,Z 369.935,A -85,B 0,C 180,E1 -16144.422,E2 -16144.422} C_VEL
LIN {X 0,Y 305.085,Z 366.925,A -85,B 0,C 180,E1 -16144.693,E2 -16144.693} C_VEL
LIN {X 0,Y 305.241,Z 364.392,A -85,B 0,C 180,E1 -16148.479,E2 -16148.479} C_VEL
LIN {X 0,Y 305.269,Z 363.089,A -85,B 0,C 180,E1 -16150.559,E2 -16150.559} C_VEL
LIN {X 0,Y 305.378,Z 363.068,A -85,B 0,C 180,E1 -16153.663,E2 -16153.663} C_VEL
LIN {X 0,Y 305.453,Z 363.064,A -85,B 0,C 180,E1 -16157.414,E2 -16157.414} C_VEL
LIN {X 0,Y 305.493,Z 363.056,A -85,B 0,C 180,E1 -16161.6,E2 -16161.6} C_VEL
LIN {X 0,Y 305.461,Z 363.06,A -85,B 0,C 180,E1 -16164.886,E2 -16164.886} C_VEL
LIN {X 0,Y 305.451,Z 363.054,A -85,B 0,C 180,E1 -16168.354,E2 -16168.354} C_VEL
LIN {X 0,Y 305.519,Z 363.047,A -85,B 0,C 180,E1 -16171.114,E2 -16171.114} C_VEL
LIN {X 0,Y 305.515,Z 363.043,A -85,B 0,C 180,E1 -16174.77,E2 -16174.77} C_VEL
LIN {X 0,Y 305.498,Z 363.038,A -85,B 0,C 180,E1 -16178.403,E2 -16178.403} C_VEL
LIN {X 0,Y 305.568,Z 363.026,A -85,B 0,C 180,E1 -16180.5,E2 -16180.5} C_VEL
LIN {X 0,Y 304.98,Z 363.113,A -85,B 0,C 180,E1 -16181.6,E2 -16181.6} C_VEL
LIN {X 0,Y 302.125,Z 363.477,A -85,B 0,C 180,E1 -16183.391,E2 -16183.391} C_VEL
LIN {X 0,Y 299.664,Z 363.773,A -85,B 0,C 180,E1 -16184.844,E2 -16184.844} C_VEL
LIN {X 0,Y 298.623,Z 363.889,A -85,B 0,C 180,E1 -16185.97,E2 -16185.97} C_VEL
LIN {X 0,Y 298.55,Z 363.895,A -85,B 0,C 180,E1 -16186.352,E2 -16186.352} C_VEL
LIN {X 0,Y 298.758,Z 363.897,A -85,B 0,C 180,E1 -16191.114,E2 -16191.114} C_VEL
LIN {X 0,Y 298.796,Z 363.891,A -85,B 0,C 180,E1 -16193.246,E2 -16193.246} C_VEL
LIN {X 0,Y 298.922,Z 363.876,A -85,B 0,C 180,E1 -16198.653,E2 -16198.653} C_VEL
LIN {X 0,Y 298.922,Z 363.877,A -85,B 0,C 180,E1 -16201.347,E2 -16201.347} C_VEL
LIN {X 0,Y 298.796,Z 363.892,A -85,B 0,C 180,E1 -16206.754,E2 -16206.754} C_VEL
LIN {X 0,Y 298.678,Z 363.906,A -85,B 0,C 180,E1 -16209.48,E2 -16209.48} C_VEL
LIN {X 0,Y 298.55,Z 363.92,A -85,B 0,C 180,E1 -16213.615,E2 -16213.615} C_VEL
LIN {X 0,Y 298.546,Z 363.92,A -85,B 0,C 180,E1 -16216.409,E2 -16216.409} C_VEL
LIN {X 0,Y 298.509,Z 363.928,A -85,B 0,C 180,E1 -16219.655,E2 -16219.655} C_VEL
LIN {X 0,Y 298.455,Z 363.936,A -85,B 0,C 180,E1 -16223.598,E2 -16223.598} C_VEL
LIN {X 0,Y 298.487,Z 363.933,A -85,B 0,C 180,E1 -16226.574,E2 -16226.574} C_VEL
LIN {X 0,Y 298.457,Z 364.082,A -85,B 0,C 180,E1 -16230.612,E2 -16230.612} C_VEL
LIN {X 0,Y 299.023,Z 367.521,A -85,B 0,C 180,E1 -16234.654,E2 -16234.654} C_VEL
LIN {X 0,Y 299.458,Z 370.26,A -85,B 0,C 180,E1 -16237.603,E2 -16237.603} C_VEL
LIN {X 0,Y 300.14,Z 374.143,A -85,B 0,C 180,E1 -16241.471,E2 -16241.471} C_VEL
LIN {X 0,Y 300.823,Z 378.547,A -85,B 0,C 180,E1 -16245.503,E2 -16245.503} C_VEL
LIN {X 0,Y 300.86,Z 381.938,A -85,B 0,C 180,E1 -16248.375,E2 -16248.375} C_VEL
LIN {X 0,Y 300.221,Z 386.054,A -85,B 0,C 180,E1 -16251.659,E2 -16251.659} C_VEL
LIN {X 0,Y 299.649,Z 389.927,A -85,B 0,C 180,E1 -16254.633,E2 -16254.633} C_VEL
LIN {X 0,Y 300.559,Z 393.131,A -85,B 0,C 180,E1 -16254.854,E2 -16254.854} C_VEL
LIN {X 0,Y 305.138,Z 405.999,A -85,B 0,C 180,E1 -16255.941,E2 -16255.941} C_VEL
LIN {X 0,Y 308.853,Z 419.208,A -85,B 0,C 180,E1 -16257.12,E2 -16257.12} C_VEL
LIN {X 0,Y 311.771,Z 433.018,A -85,B 0,C 180,E1 -16258.44,E2 -16258.44} C_VEL
LIN {X 0,Y 313.655,Z 446.202,A -85,B 0,C 180,E1 -16259.816,E2 -16259.816} C_VEL
LIN {X 0,Y 314.393,Z 455.176,A -85,B 0,C 180,E1 -16260.841,E2 -16260.841} C_VEL
LIN {X 0,Y 312.063,Z 467.514,A -85,B 0,C 180,E1 -16262.141,E2 -16262.141} C_VEL
LIN {X 0,Y 309.451,Z 479.79,A -85,B 0,C 180,E1 -16263.714,E2 -16263.714} C_VEL
LIN {X 0,Y 307.108,Z 490.129,A -85,B 0,C 180,E1 -16265.315,E2 -16265.315} C_VEL
LIN {X 0,Y 304.48,Z 501.408,A -85,B 0,C 180,E1 -16267.41,E2 -16267.41} C_VEL
LIN {X 0,Y 302.371,Z 511.063,A -85,B 0,C 180,E1 -16269.596,E2 -16269.596} C_VEL
LIN {X 0,Y 300.366,Z 519.68,A -85,B 0,C 180,E1 -16271.94,E2 -16271.94} C_VEL
LIN {X 0,Y 298.865,Z 527.049,A -85,B 0,C 180,E1 -16274.381,E2 -16274.381} C_VEL
LIN {X 0,Y 297.719,Z 533.544,A -85,B 0,C 180,E1 -16277.041,E2 -16277.041} C_VEL
LIN {X 0,Y 296.95,Z 538.779,A -85,B 0,C 180,E1 -16279.776,E2 -16279.776} C_VEL
LIN {X 0,Y 296.714,Z 541.819,A -85,B 0,C 180,E1 -16281.83,E2 -16281.83} C_VEL
LIN {X 0,Y 296.599,Z 544.784,A -85,B 0,C 180,E1 -16284.562,E2 -16284.562} C_VEL
LIN {X 0,Y 296.596,Z 546.554,A -85,B 0,C 180,E1 -16287.284,E2 -16287.284} C_VEL
LIN {X 0,Y 296.67,Z 547.162,A -85,B 0,C 180,E1 -16290.001,E2 -16290.001} C_VEL
LIN {X 0,Y 296.599,Z 546.545,A -85,B 0,C 180,E1 -16292.717,E2 -16292.717} C_VEL
LIN {X 0,Y 296.701,Z 544.448,A -85,B 0,C 180,E1 -16295.813,E2 -16295.813} C_VEL
LIN {X 0,Y 296.716,Z 541.79,A -85,B 0,C 180,E1 -16298.171,E2 -16298.171} C_VEL
LIN {X 0,Y 297.074,Z 537.564,A -85,B 0,C 180,E1 -16300.91,E2 -16300.91} C_VEL
LIN {X 0,Y 297.946,Z 531.985,A -85,B 0,C 180,E1 -16303.644,E2 -16303.644} C_VEL
LIN {X 0,Y 299.302,Z 524.904,A -85,B 0,C 180,E1 -16306.367,E2 -16306.367} C_VEL
